(* Action Save NovRAM *)
	IF xAction_SaveNovRAM OR xAction_SaveNovRAMWithoutConfirm THEN
		(* Step saving NovRAM *)
		CASE iStepActionNovRam OF
		(* check NovRAM *)
		1:	xTmp:=	T_NovRAM.T_Ctrle.xDone
					AND NOT(T_NovRAM.T_Ctrle.xExecute)
					AND NOT(T_NovRAM.T_Ctrle.xErr);
			IF xTmp THEN
				(* next Step *)
				iStepActionNovRam :=10;
				xStepActionDone:=FALSE;
			(* activ error *)
			ELSE iStepActionNovRam:=95; END_IF
		(* copy value *)
		10:	IF  xAction_SaveNovRAM THEN
				(* saving with confirmation *)
				TimerAction(IN:=FALSE);
				tTimeOutAction:=T#6s;
				T_Visu.ptrT_ExchgParam^.T_Visu.T_Message.iState:=108;	(* Confirm saving action <Enter>, or escape <Esc> ? *)
				(* next Step *)
				iStepActionNovRam :=20;
			ELSE
				(* next Step *)
				IF xAction_LoadProfileToProcessImage OR xAction_SaveProfileToFile OR xActionDeleteProfile  THEN
					IF xAction_LoadProfileToProcessImage THEN
						T_NovRam.T_Data.T_Standard.T_InfoProcess.iProfile:=T_VisuQVis.ptrT_ExchgParam^.T_StationCommon.T_InfoProcess.iProfile;
						T_NovRam.T_Data.T_Standard.T_InfoProcess.sProfileName:=T_VisuQVis.ptrT_ExchgParam^.T_StationCommon.T_InfoProcess.sProfileName;
					END_IF;
					iStepActionNovRam :=40;
				ELSE
					iStepActionNovRam :=30;
				END_IF;
				(* Display message *)
				T_Visu.ptrT_ExchgParam^.T_Visu.T_Message.iState:=13;	(* Start saving *)
			END_IF;
		(* waiting for saving confirmation key <Enter> or <Esc> *)
		20:	IF RisingEdgeKeyPanel_Enter.Q THEN
			(* Display message *)
				T_Visu.ptrT_ExchgParam^.T_Visu.T_Message.iState:=13;	(* Start saving *)
				(* next step *)
				iStepActionNovRam:=30;
			ELSE
				IF RisingEdgeKeyPanel_Esc.Q THEN iStepActionNovRam:=60; END_IF
				(* An other message has been displayed, stop saving action *)
				IF T_Visu.ptrT_ExchgParam^.T_Visu.T_Message.iState<>108 THEN iStepActionNovRam:=60; END_IF
			END_IF
		30:	T_NovRAM.T_Data.T_ProcessImageData.T_GeometryPara:=T_Visu.ptrT_ExchgParam^.T_GeometryCommon.T_Geometry;
			T_NovRAM.T_Data.T_ProcessImageData.T_PrismPara:=T_Visu.ptrT_ExchgParam^.T_StationCommon.T_PrismPara;
			IF (T_NovRAM.T_Data.T_ProcessImageData.T_PrismPara.bStateInputPrisma = 1) THEN
				T_NovRAM.T_Data.T_ProcessImageData.T_PrismPara.bStateInputPrisma:=0;
			END_IF;
			IF (T_NovRAM.T_Data.T_ProcessImageData.T_PrismPara.bStateInputPrisma = 3) THEN
				T_NovRAM.T_Data.T_ProcessImageData.T_PrismPara.bStateInputPrisma:=2;
			END_IF;
			rCalcMinMaxToolDia:=	rFctCalcMaxToolDiameter(	rDistanceD1:=T_NovRAM.T_Data.T_ProcessImageData.T_PrismPara.rPrismaDistanceD1,
														rDistanceD2:=T_NovRAM.T_Data.T_ProcessImageData.T_PrismPara.rPrismaDistanceD2,
														rAnglePrism:=T_NovRAM.T_Data.T_ProcessImageData.T_PrismPara.rPrismaAngleA);
			T_NovRAM.T_Data.T_ProcessImageData.T_PrismPara.rToolDiameterMax:=rCalcMinMaxToolDia;
			rCalcMinMaxToolDia:=	rFctCalcMinToolDiameter(	rDistanceD1:=T_NovRAM.T_Data.T_ProcessImageData.T_PrismPara.rPrismaDistanceD1,
														rDistanceD2:=T_NovRAM.T_Data.T_ProcessImageData.T_PrismPara.rPrismaDistanceD2,
														rAnglePrism:=T_NovRAM.T_Data.T_ProcessImageData.T_PrismPara.rPrismaAngleA,
														bStateInputPrisma:=T_NovRAM.T_Data.T_ProcessImageData.T_PrismPara.bStateInputPrisma);
			T_NovRAM.T_Data.T_ProcessImageData.T_PrismPara.rToolDiameterMin:=rCalcMinMaxToolDia;
			rCalcPrismaFactor:=	rFctCalcPrismaFactor(	rAnglePrism:=T_NovRAM.T_Data.T_ProcessImageData.T_PrismPara.rPrismaAngleA);
			T_NovRAM.T_Data.T_ProcessImageData.T_PrismPara.rPrismaFactor:=rCalcPrismaFactor;
			T_Visu.ptrT_ExchgParam^.T_StationCommon.T_PrismPara:=T_NovRAM.T_Data.T_ProcessImageData.T_PrismPara;
			T_NovRAM.T_Data.T_Standard.T_TeachINToolLeft:=T_Visu.ptrT_ExchgParam^.T_TeachIn.TParam_ToolLeft;
			T_NovRAM.T_Data.T_Standard.T_TeachINToolCenter:=T_Visu.ptrT_ExchgParam^.T_TeachIn.TParam_ToolCenter;
			T_NovRAM.T_Data.T_Standard.T_TeachINToolRight:=T_Visu.ptrT_ExchgParam^.T_TeachIn.TParam_ToolRight;
			T_NovRAM.T_Data.T_Standard.T_TeachINToolFeeder:=T_Visu.ptrT_ExchgParam^.T_TeachIn.TParam_ToolFeeder;
			T_NovRAM.T_Data.T_Standard.T_TeachINGrindFeeder:=T_Visu.ptrT_ExchgParam^.T_TeachIn.TParam_GrindFeeder;
			T_NovRAM.T_Data.T_Standard.T_AxisPosition:=T_Visu.ptrT_ExchgParam^.T_TeachIn.TParam_AxisPosition;
			T_NovRAM.T_Data.T_Standard.T_MachineConfig.iConfigMachineType:=T_Visu.ptrT_ExchgParam^.T_StationCommon.iConfigMachineType;
			T_NovRAM.T_Data.T_Standard.T_MachineConfig.iConfigAxisType:=T_Visu.ptrT_ExchgParam^.T_StationCommon.iConfigAxisType;
			T_NovRAM.T_Data.T_Standard.T_MachineConfig.iConfigVisuNavigation:=T_Visu.ptrT_ExchgParam^.T_StationCommon.iConfigVisuNavigation;
			T_NovRAM.T_Data.T_Standard.T_MachineConfig.rConfigMaxToolLength:=T_Visu.ptrT_ExchgParam^.T_StationCommon.rConfigMaxToolLength;
			T_NovRAM.T_Data.T_Standard.T_ToolTensionSystem:=T_Visu.ptrT_ExchgParam^.T_StationCommon.T_ParamToolTensionSystem;
			T_NovRAM.T_Data.T_Standard.T_Cyl_ToolTension:=T_Visu.ptrT_ExchgParam^.T_Cylinder.T_ParamToolTension;
			T_NovRAM.T_Data.T_ProcessImageData.T_AutoGeometryPara:=T_Visu.ptrT_ExchgParam^.T_StationCommon.T_AutoGeometryPara;
			T_NovRAM.T_Data.T_ProcessImageData.T_AutoGroovePara:=T_Visu.ptrT_ExchgParam^.T_StationCommon.T_AutoGroovePara;
			T_NovRAM.T_Data.T_ProcessImageData.T_CalibrationPara:=T_Visu.ptrT_ExchgParam^.T_StationCommon.T_CalibrationPara;
			T_NovRAM.T_Data.T_ProcessImageData.T_ProcessPara:=T_Visu.ptrT_ExchgParam^.T_StationCommon.T_ProcessPara;
			(* next Step *)
			iStepActionNovRam :=40;
		(* activ save *)
		40:	T_NovRAM.T_Ctrle.xExecute:=TRUE;
			T_NovRAM.T_Ctrle.iFunction:=2;
			(* next Step *)
			iStepActionNovRam :=50;
			xStepActionDone:=FALSE;
		(* wait save confirmation *)
		50:	IF NOT(xStepActionDone) THEN
				T_NovRAM.T_Ctrle.xExecute:=FALSE;
				(* confirm Step *)
				xStepActionDone:=TRUE;
			ELSE
				IF T_NovRAM.T_Ctrle.xDone THEN
				(* next Step *)
					IF (T_Visu.T_PlcParam.dwActualPage = 430) OR ((T_Visu.T_PlcParam.dwActualPage = 130) AND (T_Visu.T_CtrleAction.iFunction = 1002)) OR
					     ((T_Visu.T_PlcParam.dwActualPage = 470) AND (T_Visu.ptrT_ExchgParam^.T_Config.iEditParam = 410)) THEN
						iStepActionNovRam :=51;
						xOpenMessageBox:=FALSE;
					ELSE
						iStepActionNovRam :=90;
					END_IF;
					xStepActionDone:=FALSE;
				ELSE	IF T_NovRAM.T_Ctrle.xErr THEN
							iStepActionNovRam:=99;
							xStepActionDone:=FALSE;
						END_IF
				END_IF
			END_IF
		(* check first if the Actual position is between the pos and neg SW limit switch *)
		51:	IF (T_Station.THardware.TAxisGrindFeeder.T_LiveValue.lrActualPosition >= T_NovRAM.T_Data.T_ProcessImageData.T_PrismPara.rToolDiameterMin) AND
			     (T_Station.THardware.TAxisGrindFeeder.T_LiveValue.lrActualPosition <= (T_NovRAM.T_Data.T_ProcessImageData.T_PrismPara.rToolDiameterMax + T_NovRAM.T_Data.T_Standard.T_TeachINGrindFeeder.rOffsetSWPosEndSwitch)) THEN
				(* Actual Position is not over the SW limit switches *)
				iStepActionNovRam :=53;
			ELSE
				(* Actual Position is over the SW limit switches *)
				T_Station.THardware.TAxisGrindFeeder.T_CtrleSingle.iFunction:=29;		(* Switch off the SW limit switches, in this case the GrindFeeder will not move automatically *)
				T_Station.THardware.TAxisGrindFeeder.T_CtrleSingle.xExecute:=TRUE;
				iStepActionNovRam :=52;
				xOpenMessageBox:=TRUE;
				tTimeOutAction:=tTimeOutAction + T#9999s;
			END_IF;
		(* Wait end of resettet SW end switch for the GrindFeeder Axis *)
		52:	IF NOT(T_Station.THardware.TAxisGrindFeeder.T_CtrleSingle.xExecute) AND T_Station.THardware.TAxisGrindFeeder.T_CtrleSingle.xDone THEN
				(* set the new position of the GrindFeeder Axis *)
				T_Station.THardware.TAxisGrindFeeder.T_CtrleSingle.rSetPosition:=T_NovRAM.T_Data.T_ProcessImageData.T_PrismPara.rToolDiameterMin;
				T_Station.THardware.TAxisGrindFeeder.T_CtrleSingle.iFunction:=11;
				T_Station.THardware.TAxisGrindFeeder.T_CtrleSingle.xExecute:=TRUE;
				lrActualGrindFeedPosition:=DINT_TO_LREAL(LREAL_TO_DINT(T_Station.THardware.TAxisGrindFeeder.T_LiveValue.lrActualPosition * 100.0)) / 100.0;
				lrToWriteGrindFeedPosition:=DINT_TO_LREAL(LREAL_TO_DINT(T_NovRAM.T_Data.T_ProcessImageData.T_PrismPara.rToolDiameterMin * 100.0)) / 100.0;
				iStepActionNovRam :=53;
			END_IF;
			IF NOT(T_Station.THardware.TAxisGrindFeeder.T_CtrleSingle.xExecute) AND T_Station.THardware.TAxisGrindFeeder.T_CtrleSingle.xErr THEN
				iStepActionNovRam :=98;
			END_IF;
		(* Set SW end switch for the GrindFeeder Axis *)
		53:	IF NOT(T_Station.THardware.TAxisGrindFeeder.T_CtrleSingle.xExecute) AND T_Station.THardware.TAxisGrindFeeder.T_CtrleSingle.xDone THEN
				T_Station.THardware.TAxisGrindFeeder.T_CtrleSingle.iFunction:=28;
				T_Station.THardware.TAxisGrindFeeder.T_CtrleSingle.lrSWNegLimitSwitch:=T_NovRAM.T_Data.T_ProcessImageData.T_PrismPara.rToolDiameterMin;
				T_Station.THardware.TAxisGrindFeeder.T_CtrleSingle.lrSWPosLimitSwitch:=T_NovRAM.T_Data.T_ProcessImageData.T_PrismPara.rToolDiameterMax + T_NovRAM.T_Data.T_Standard.T_TeachINGrindFeeder.rOffsetSWPosEndSwitch;
				T_Station.THardware.TAxisGrindFeeder.T_CtrleSingle.xExecute:=TRUE;
				iStepActionNovRam :=54;
			END_IF;
			IF NOT(T_Station.THardware.TAxisGrindFeeder.T_CtrleSingle.xExecute) AND T_Station.THardware.TAxisGrindFeeder.T_CtrleSingle.xErr THEN
				iStepActionNovRam :=98;
			END_IF;
		(* Wait end of settled SW end switch for the GrindFeeder Axis *)
		54:	IF NOT(T_Station.THardware.TAxisGrindFeeder.T_CtrleSingle.xExecute) AND T_Station.THardware.TAxisGrindFeeder.T_CtrleSingle.xDone THEN
				IF xOpenMessageBox THEN
					xOpenMessageBox:=FALSE;
					iStepActionNovRam :=55;
				ELSE
					iStepActionNovRam :=90;
				END_IF;
			END_IF;
			IF NOT(T_Station.THardware.TAxisGrindFeeder.T_CtrleSingle.xExecute) AND T_Station.THardware.TAxisGrindFeeder.T_CtrleSingle.xErr THEN
				iStepActionNovRam :=98;
			END_IF;
		(* Open MessageBox *)
		55:	T_Visu.ptrT_ExchgParam^.T_FunctionCommon.sMessageBoxLine1:='The prisma value are changed and the actual ';
			T_Visu.ptrT_ExchgParam^.T_FunctionCommon.sMessageBoxLine2:='GrindFeeder position is now over the';
			T_Visu.ptrT_ExchgParam^.T_FunctionCommon.sMessageBoxLine3:='Software limit switches. The actual absolut';
			T_Visu.ptrT_ExchgParam^.T_FunctionCommon.sMessageBoxLine4:='GrindFeeder position: ';
			T_Visu.ptrT_ExchgParam^.T_FunctionCommon.sMessageBoxLine4:=CONCAT(T_Visu.ptrT_ExchgParam^.T_FunctionCommon.sMessageBoxLine4,
																				LREAL_TO_STRING(lrActualGrindFeedPosition));
			T_Visu.ptrT_ExchgParam^.T_FunctionCommon.sMessageBoxLine4:=CONCAT(T_Visu.ptrT_ExchgParam^.T_FunctionCommon.sMessageBoxLine4,'um');
			T_Visu.ptrT_ExchgParam^.T_FunctionCommon.sMessageBoxLine5:='is overwritten with the minimum ';
			T_Visu.ptrT_ExchgParam^.T_FunctionCommon.sMessageBoxLine6:='ToolDiameter: ';
			T_Visu.ptrT_ExchgParam^.T_FunctionCommon.sMessageBoxLine6:=CONCAT(T_Visu.ptrT_ExchgParam^.T_FunctionCommon.sMessageBoxLine6,
																				LREAL_TO_STRING(lrToWriteGrindFeedPosition));
			T_Visu.ptrT_ExchgParam^.T_FunctionCommon.sMessageBoxLine6:=CONCAT(T_Visu.ptrT_ExchgParam^.T_FunctionCommon.sMessageBoxLine6,'um');
			T_Visu.ptrT_ExchgParam^.T_FunctionCommon.xOpenOverlayMessageBox:=TRUE;
			iStepActionNovRam :=56;
		(* Wait cofirming of the messagebox *)
		56:	IF NOT(T_Visu.ptrT_ExchgParam^.T_FunctionCommon.xOpenOverlayMessageBox) THEN
				iStepActionNovRam :=90;
			END_IF;
			IF T_Visu.T_CtrleAction.xDone THEN
				T_Visu.ptrT_ExchgParam^.T_FunctionCommon.xOpenOverlayMessageBox:=FALSE;
				xAction_SaveNovRAM:=FALSE;
				xAction_SaveNovRAMWithoutConfirm:=FALSE;
				T_Visu.ptrT_ExchgParam^.T_Visu.T_Message.iState:=0;
			END_IF;
		(* Reset settled value *)
		60:	xResetParaListValue:=TRUE;
			iStepActionNovRam:=70;
		70:	IF NOT(xResetParaListValue) THEN
				iStepActionNovRam:=90;
			END_IF;
		(* no code, waiting timeout *)
		89:	IF TimerAction.Q THEN iStepActionNovRam:=90; END_IF
		(* save done *)
		90:	T_Visu.ptrT_ExchgParam^.T_Visu.T_Message.iState:=0;
			T_Visu.T_CtrleAction.xDone:=TRUE;
			T_Visu.T_CtrleAction.xNotReady:=FALSE;
			T_Visu.T_CtrleAction.xErr:=FALSE;
			T_Visu.T_CtrleAction.udiErrorID:=0;
			xAction_SaveNovRAM:=FALSE;
			xAction_SaveNovRAMWithoutConfirm:=FALSE;
			T_Visu.ptrT_ExchgParam^.T_FunctionCommon.xOpenOverlayMessageBox:=FALSE;
		(* NovRAM not ready *)
		95:	TimerNotReady(IN:=TRUE);
			xAction_SaveNovRAM:=FALSE;
			xAction_SaveNovRAMWithoutConfirm:=FALSE;
			T_Visu.ptrT_ExchgParam^.T_FunctionCommon.xOpenOverlayMessageBox:=FALSE;
		(* error *)
		98:	T_Visu.ptrT_ExchgParam^.T_StationCommon.wState:=T_Visu.ptrT_ExchgParam^.T_StationCommon.wState AND 16#BF;
			T_Visu.T_CtrleAction.xDone:=TRUE;
			T_Visu.T_CtrleAction.xNotReady:=FALSE;
			IF (T_Station.THardware.TAxisGrindFeeder.T_Config_Gen.iTyp <> 0) THEN
				diErrorNr:=(T_Station.THardware.TAxisGrindFeeder.T_Config_Gen.iTyp * 1000000) + T_Station.THardware.TAxisGrindFeeder.T_CtrleSingle.udiErrorID;
			ELSE
				diErrorNr:=0;
			END_IF;
			FBErrorMessage(	diErrorNr:=diErrorNr,
							T_ErrorList:=T_ErrorList);
			T_Visu.ptrT_ExchgParam^.T_Visu.T_Message.sDynamicTextEnglish:=FBErrorMessage.sErrorTextEnglish;
			T_Visu.ptrT_ExchgParam^.T_Visu.T_Message.sDynamicTextDeutsch:=FBErrorMessage.sErrorTextDeutsch;
			T_Visu.ptrT_ExchgParam^.T_Visu.T_Message.sDynamicTextFrancais:=FBErrorMessage.sErrorTextFrancais;
			T_Visu.ptrT_ExchgParam^.T_SafetyCtrl.xSetForceError:=TRUE;
			T_Visu.ptrT_ExchgParam^.T_SafetyCtrl.diSetForceErrorNr:=diErrorNr;
			T_Visu.T_CtrleAction.xErr:=FALSE;
			T_Visu.T_CtrleAction.udiErrorID:=0;
			T_Station.THardware.TAxisGrindFeeder.T_CtrleSingle.iFunction:=1;
			T_Station.THardware.TAxisGrindFeeder.T_CtrleSingle.xExecute:=TRUE;
			xAction_SaveNovRAM:=FALSE;
			xAction_SaveNovRAMWithoutConfirm:=FALSE;
			T_Visu.ptrT_ExchgParam^.T_FunctionCommon.xOpenOverlayMessageBox:=FALSE;
		(* error *)
		99:	T_Visu.T_CtrleAction.xDone:=FALSE;
			T_Visu.T_CtrleAction.xNotReady:=FALSE;
			T_Visu.T_CtrleAction.xErr:=TRUE;
			T_Visu.T_CtrleAction.udiErrorID:=16#F0000 + T_Visu.T_CtrleAction.iFunction;
			xAction_SaveNovRAM:=FALSE;
			xAction_SaveNovRAMWithoutConfirm:=FALSE;
			T_Visu.ptrT_ExchgParam^.T_FunctionCommon.xOpenOverlayMessageBox:=FALSE;
		END_CASE
	END_IF;

(* Delete Profile *)
	IF xActionDeleteProfile THEN
		(* Step delete profile *)
		CASE iStepAction OF
		(* Profile number could not be 1 *)
		1:	IF T_Visu.ptrT_ExchgParam^.T_ProfileCommon.T_Id.iNumber < 2 THEN
				 tTimeOutAction:=TimerAction.ET+T#2s;
				T_Visu.ptrT_ExchgParam^.T_Visu.T_Message.iState:=27;	(* Default profile can't be deleted *)
				iStepAction:=10;
			ELSIF T_Visu.ptrT_ExchgParam^.T_StationCommon.T_InfoProcess.iProfile = T_Visu.ptrT_ExchgParam^.T_ProfileCommon.T_Id.iNumber THEN
				tTimeOutAction:=TimerAction.ET+T#2s;
				T_Visu.ptrT_ExchgParam^.T_Visu.T_Message.iState:=28;	(* Load profile can't be deleted *)
				iStepAction:=10;
			ELSE iStepAction:=20; END_IF
		(* no code, waiting timeout *)
		10:	IF TimerAction.Q THEN xActionDeleteProfile:=FALSE; END_IF;
		(* Display message to ask for confirmation *)
		20:	T_Visu.ptrT_ExchgParam^.T_Visu.T_Message.iState:=117;	(* Confirm delete profile <Enter>, or escape <Esc> ? *)
			(* next step *)
			iStepAction:=30;
		(* waiting for key <Enter> or <Esc> *)
		30:	IF RisingEdgeKeyPanel_Enter.Q THEN
				(* Display message deleting *)
				T_Visu.ptrT_ExchgParam^.T_Visu.T_Message.iState:=29;	(* Start deleting *)
				(* next step *)
				iStepAction:=40;
			ELSE
				IF RisingEdgeKeyPanel_Esc.Q THEN iStepAction:=90; END_IF
				(* An other message has been displayed, stop import/export action *)
				IF T_Visu.ptrT_ExchgParam^.T_Visu.T_Message.iState<>117 THEN iStepAction:=90; END_IF
			END_IF;
		(* Init. deleting profile file *)
		40:	IF T_NovRam.T_Data.T_IDProfileStation[T_Visu.ptrT_ExchgParam^.T_ProfileCommon.T_Id.iNumber].sName <> '' THEN
				sTmp:='\Hard Disk\Machine450\Profile\';
				sTmp:=CONCAT(sTmp,T_NovRam.T_Data.T_IDProfileStation[T_Visu.ptrT_ExchgParam^.T_ProfileCommon.T_Id.iNumber].sName);
				T_HDD.T_File.sPathAndFileName:=CONCAT(sTmp,'.txt');
				(* activ delete file *)
				T_HDD.T_Ctrle.xExecute:=TRUE;
				T_HDD.T_Ctrle.iFunction:=5;
				iStepAction:=50;
			(* Display info message 'file does not exists *)
			ELSE
				T_Visu.ptrT_ExchgParam^.T_Visu.T_Message.iState:=11;
				(* next step *)
				iStepAction:=55;
				xStepActionDone:=FALSE;
				tTimeOutAction:=TimerAction.ET+T#2s;
			END_IF
		50:	IF NOT T_HDD.T_Ctrle.xExecute AND (T_HDD.T_Ctrle.xDone OR T_HDD.T_Ctrle.xErr) THEN
				T_HDD.T_Ctrle.xReset:=T_HDD.T_Ctrle.xErr;
				(* Profile will be erased from the profile list *)
				T_NovRam.T_Data.T_IDProfileStation[T_Visu.ptrT_ExchgParam^.T_ProfileCommon.T_Id.iNumber].sName:='';
				xUpdateProfileList:=TRUE;
				IF T_HDD.T_Ctrle.xErr THEN
					(* Display info message 'file does not exists *)
					T_Visu.ptrT_ExchgParam^.T_Visu.T_Message.iState:=11;
					(* next step *)
					iStepAction:=52;
					xStepActionDone:=FALSE;
					(* use tmp timer to diplay message *)
					TimerONTmp(IN:=FALSE);
					TimerONTmp.PT:=T#2s;
				ELSE
					(* next step *)
					iStepAction:=70;
					xStepActionDone:=FALSE;
				END_IF;
			END_IF
		(* Wait delay timer *)
		52:	IF TimerONTmp.Q THEN
				T_Visu.ptrT_ExchgParam^.T_Visu.T_Message.iState:=0;
				(* next step *)
				iStepAction:=70;
			END_IF
		(* delay time out *)
		55:	IF TimerAction.Q THEN xActionDeleteProfile:=FALSE; END_IF
		(* active saving data NovRAM *)
		70:	T_Visu.ptrT_ExchgParam^.T_ProfileCommon.T_Id.sName:='';
			xAction_SaveNovRAMWithoutConfirm:=TRUE;
			iStepActionNovRam:=1;
			(* next step *)
			iStepAction:=80;
		(* waiting confirm saving NovRAM action *)
		80:	IF NOT xAction_SaveNovRAMWithoutConfirm THEN iStepAction:=90; END_IF
		(* save done *)
		90:	T_Visu.ptrT_ExchgParam^.T_Visu.T_Message.iState:=0;
			T_Visu.T_CtrleAction.xDone:=TRUE;
			T_Visu.T_CtrleAction.xNotReady:=FALSE;
			T_Visu.T_CtrleAction.xErr:=FALSE;
			T_Visu.T_CtrleAction.udiErrorID:=0;
			xActionDeleteProfile:=FALSE;
		(* Action not ready *)
		95:	TimerNotReady(IN:=TRUE);
			xActionDeleteProfile:=FALSE;
		(* error *)
		99:	T_Visu.T_CtrleAction.xDone:=FALSE;
			T_Visu.T_CtrleAction.xNotReady:=FALSE;
			T_Visu.T_CtrleAction.xErr:=TRUE;
			T_Visu.T_CtrleAction.udiErrorID:=16#F1000 + T_Profile.T_Ctrle.iFunction;
			xActionDeleteProfile:=FALSE;
		END_CASE;
	END_IF;

(* Action start process machine or station *)
	IF xActionProcMachine OR xActionProcStation THEN
		(* Step process machine *)
		CASE iStepAction OF
		(* check process state *)
		1:	xTmp:=	T_Process.xEnable AND
					T_Process.xEnd AND
					T_Process.xRdy AND
					NOT(T_Process.xStop) AND
					NOT(T_Process.xStopCycle) AND
					NOT(T_Process.xError);
			(* next step *)
			IF NOT(xTmp) THEN
				iStepAction:=95;
			ELSE IF xActionProcMachine THEN iStepAction:=10; ELSE iStepAction:=20; END_IF
			END_IF
		(* check process number and start process machine *)
		10:	CASE T_Process.iFunctNr OF
			(* process available *)
			(*	10=Process AutoGeometry
				20=Process AutoGroove
				30=Process Reference
			*)
			10,20,30:	T_Visu.T_CtrleProcess.iFunction:=1;
						T_Visu.T_CtrleProcess.xExecute:=TRUE;
						iStepAction:=90;
			(* unknown process *)
			ELSE	iStepAction:=95;
			END_CASE
			(* next step *)
			xStepActionDone:=FALSE;
		(* check process number and start process station *)
		20:	CASE T_Process.iFunctNr OF
			(* process available *)
			(*	40=ToolCalibration
			*)
			40:	T_Visu.T_CtrleProcess.iFunction:=2;
				T_Visu.T_CtrleProcess.xExecute:=TRUE;
				iStepAction:=90;
			(* unknown process *)
			ELSE
				iStepAction:=95;
			END_CASE
			(* next step *)
			xStepActionDone:=FALSE;
		(* Display message, waiting timeout *)
		89:	IF TimerAction.Q THEN
				(* init. trigger FB_CtrleButton Start/Stop *)
				T_Visu.ptrT_ExchgParam^.T_Machine.T_Process.wState:=16#0;
				(* action done *)
				iStepAction:=90;
			END_IF
		(* action done *)
		90:	T_Visu.T_CtrleAction.xDone:=TRUE;
			T_Visu.T_CtrleAction.xNotReady:=FALSE;
			T_Visu.T_CtrleAction.xErr:=FALSE;
			T_Visu.T_CtrleAction.udiErrorID:=0;
			xActionProcMachine:=FALSE;
			xActionProcStation:=FALSE;
		(* cylinder not ready *)
		95:	TimerNotReady(IN:=TRUE);
			xActionProcMachine:=FALSE;
			xActionProcStation:=FALSE;
		(* error *)
		99:	T_Visu.T_CtrleAction.xDone:=FALSE;
			T_Visu.T_CtrleAction.xNotReady:=FALSE;
			T_Visu.T_CtrleAction.xErr:=TRUE;
			T_Visu.T_CtrleAction.udiErrorID:=16#F0000 + T_Visu.T_CtrleAction.iFunction;
			xActionProcMachine:=FALSE;
			xActionProcStation:=FALSE;
		END_CASE
	END_IF

(* Manage process execution *)
	(* ...done *)
	RisingEdgeProcessDone(CLK:=T_Visu.T_CtrleProcess.xDone);
	IF RisingEdgeProcessDone.Q THEN
		IF NOT(T_StartUp.T_State.xBlockChangeMovementVisu) THEN
			IF T_Visu.T_CtrleProcess.iFunction <> 0 AND T_Visu.ptrT_ExchgParam^.T_Visu.T_Message.iState = 0 THEN
			(* call confirmation message *)
				IF NOT xStopImmediatly THEN
					IF (T_Visu.T_PlcParam.dwActualPage = 110) THEN
						T_Visu.ptrT_ExchgParam^.T_Visu.T_Message.iState:=22;
					END_IF;
					(*T_Visu.ptrT_ExchgParam^.T_Visu.T_Message.iState
						:=iFctReturnConfMessage(iNumAction:=T_Process.iFunctNr+1100);*);
				(* Display message 'Process is aborded' *)
				ELSE T_Visu.ptrT_ExchgParam^.T_Visu.T_Message.iState:=9; END_IF
			END_IF
		END_IF;
	END_IF
	(* ...error *)
	RisingEdgeProcessError(CLK:=T_Visu.T_CtrleProcess.xErr);
	IF RisingEdgeProcessError.Q THEN
	(* call function bloc action error *)
		IF NOT(T_StartUp.T_State.xBlockChangeMovementVisu) THEN
			(*
			fbQvisError(	udiActionError:=T_Visu.T_CtrleProcess.udiErrorID,
						T_Message:=T_Visu.ptrT_ExchgParam^.T_Visu.T_Message);
			*);
		END_IF;
		(* Init. variable *)
		T_Visu.T_CtrleProcess.xExecute:=FALSE;
		T_Visu.T_CtrleProcess.xDone:=TRUE;
		T_Visu.T_CtrleProcess.xErr:=FALSE;
		T_Visu.T_CtrleProcess.udiErrorID:=0;
		(*iStepProcess:=1;*)
		(*xStepProcessDone:=FALSE;*)
	END_IF
	(* ...reset *)
	RisingEdgeResetProcess(CLK:=T_Visu.T_CtrleProcess.xReset);
	IF RisingEdgeResetProcess.Q THEN
		(* Init. variable *)
		T_Visu.T_CtrleProcess.xExecute:=FALSE;
		T_Visu.T_CtrleProcess.xDone:=TRUE;
		T_Visu.T_CtrleProcess.xErr:=FALSE;
		T_Visu.T_CtrleProcess.udiErrorID:=0;
		(*iStepProcess:=1;*)
		(*xStepProcessDone:=FALSE;*)
		(* Release process *)
		T_Visu.T_CtrleProcess.xReset:=FALSE;
	END_IF
	RisingEdgeExecuteProcess(CLK:=T_Visu.T_CtrleProcess.xExecute);
	IF RisingEdgeExecuteProcess.Q THEN
		(* Release execution *)
		T_Visu.T_CtrleProcess.xExecute:=FALSE;
		CASE T_Visu.T_CtrleProcess.iFunction OF
		(* Process machine *)
		1:	xProcessMachine:=TRUE;
		(* Process station *)
		2:	xProcessStation:=TRUE;
		(* process not implemented *)
		ELSE	T_Visu.T_CtrleProcess.xDone:=FALSE;
				T_Visu.T_CtrleProcess.xErr:=TRUE;
				T_Visu.T_CtrleProcess.udiErrorID:=16#E000;
				(* exit FB *)
				RETURN;
		END_CASE
		(* Init. variable *)
		T_Visu.T_CtrleProcess.xDone:=FALSE;
		T_Visu.T_CtrleProcess.xErr:=FALSE;
		T_Visu.T_CtrleProcess.udiErrorID:=0;
		iStepProcess:=1;
		xStepProcessDone:=FALSE;
		(* exit FB *)
		RETURN;
	END_IF

(* Process machine *)
	IF xProcessMachine OR xProcessStation THEN
		CASE iStepProcess OF
		(* check process number and start process machine *)
		1:	T_Process.xStart:=TRUE;
			iStepProcess:=10;
			IF (T_Visu.T_PlcParam.dwActualPage = 10) THEN
				T_Visu.ptrT_ExchgParam^.T_SafetyCtrl.bStateAutoGeometry:=2;
			ELSIF (T_Visu.T_PlcParam.dwActualPage = 20) THEN
				T_Visu.ptrT_ExchgParam^.T_SafetyCtrl.bStateAutoGroove:=2;
			ELSIF (T_Visu.T_PlcParam.dwActualPage = 30) THEN
				T_Visu.ptrT_ExchgParam^.T_SafetyCtrl.bStateReference:=2;
			ELSIF (T_Visu.T_PlcParam.dwActualPage = 110) THEN
				T_Visu.ptrT_ExchgParam^.T_SafetyCtrl.bStateToolCalibration:=2;
			END_IF;
			(* next step *)
			xStepProcessDone:=FALSE;
		(* wait confirmation *)
		10:	IF NOT(xStepProcessDone) THEN
			(* release execution *)
				T_Process.xStart:=FALSE;
				xStepProcessDone:=TRUE;
				IF T_Visu.ptrT_ExchgParam^.T_StationCommon.T_AutoGeometryPara.xWarmUp THEN
					xWarmUpMessageActiv:=TRUE;
					xWarmUpMessageDone:=TRUE;
				END_IF;
			ELSE
				IF T_Process.xEnd THEN
					(* action done *)
					iStepProcess:=90;
					xStepProcessDone:=FALSE;
				ELSE
					IF T_Visu.ptrT_ExchgParam^.T_StationCommon.T_AutoGeometryPara.xWarmUp AND xWarmUpMessageActiv THEN
						T_Visu.ptrT_ExchgParam^.T_Visu.T_Message.iState:=124;	(* WarmUp cycle activ *)
						xWarmUpMessageActiv:=FALSE;
					END_IF;
					IF (T_Visu.ptrT_ExchgParam^.T_Visu.T_Message.iState=124                                                 )	AND
					     NOT(T_Visu.ptrT_ExchgParam^.T_StationCommon.T_AutoGeometryPara.xWarmUp) 	AND
					     xWarmUpMessageDone 															THEN
						T_Visu.ptrT_ExchgParam^.T_Visu.T_Message.iState:=125;	(*WarmUp cycle time arrived. <Press StopButton>*)
						xWarmUpMessageDone:=FALSE;
					END_IF;
					IF T_Process.xError THEN
						(* action error *)
						iStepProcess:=99;
						xStepProcessDone:=FALSE;
						IF xProcessMachine THEN
							T_Visu.ptrT_ExchgParam^.T_TouchScreenBtPanel.iStateBtLeft:=0;
							IF(T_Process.iFunctNr = 10) THEN
								IF (T_Visu.T_PlcParam.dwActualPage <> 10) THEN
									T_Visu.T_PlcParam.dwSetNewPage:=10;
									T_Visu.T_CtrleVisu.iFunction:=1;
									T_Visu.T_CtrleVisu.xExecute:=TRUE;
								END_IF;
							END_IF;
							IF(T_Process.iFunctNr = 20) THEN
								IF (T_Visu.T_PlcParam.dwActualPage <> 20) THEN
									T_Visu.T_PlcParam.dwSetNewPage:=20;
									T_Visu.T_CtrleVisu.iFunction:=1;
									T_Visu.T_CtrleVisu.xExecute:=TRUE;
								END_IF;
							END_IF;
							IF(T_Process.iFunctNr = 30) THEN
								IF (T_Visu.T_PlcParam.dwActualPage <> 30) THEN
									T_Visu.T_PlcParam.dwSetNewPage:=30;
									T_Visu.T_CtrleVisu.iFunction:=1;
									T_Visu.T_CtrleVisu.xExecute:=TRUE;
								END_IF;
							END_IF;
							IF(T_Process.iFunctNr = 40) THEN
								IF (T_Visu.T_PlcParam.dwActualPage <> 110) THEN
									T_Visu.T_PlcParam.dwSetNewPage:=110;
									T_Visu.T_CtrleVisu.iFunction:=1;
									T_Visu.T_CtrleVisu.xExecute:=TRUE;
								END_IF;
							END_IF;
						END_IF;
					END_IF
				END_IF
				IF NOT(T_TwinSafeOut.QxContactor_K3) OR NOT(T_TwinSafeOut.QxContactor_K4) THEN
					(*T_Process.xEnable:=FALSE;*)
					(*iStepProcess:=21;*)
					iStepProcess:=99;
					RETURN;
				END_IF;
			END_IF
		21:	IF NOT(T_Process.xEnd) THEN
				T_Process.xEnable:=TRUE;
				iStepProcess:=22;
			ELSE
				T_Process.xEnable:=FALSE;
			END_IF;
		22:	IF T_Process.xEnd THEN
				T_Visu.T_CtrleProcess.xDone:=TRUE;
				T_Visu.T_CtrleProcess.xErr:=FALSE;
				T_Visu.T_CtrleProcess.udiErrorID:=0;
				xProcessMachine:=FALSE;
				xProcessStation:=FALSE;
			END_IF;
		(* call page *)
		30:	T_Visu.T_PlcParam.dwSetNewPage:=dwPageNrProcessStart;
			T_Visu.T_CtrleVisu.iFunction:=2;
			T_Visu.T_CtrleVisu.xExecute:=TRUE;
			(* next step *)
			iStepProcess:=90;
		(* process done *)
		90:	IF NOT(T_Visu.T_CtrleVisu.xExecute) AND T_Visu.T_CtrleVisu.xDone THEN
				T_StartUp.T_State.xBlockChangeMovementVisu:=FALSE;
				IF (T_Visu.T_PlcParam.dwActualPage = 10) THEN
					T_Visu.ptrT_ExchgParam^.T_SafetyCtrl.bStateAutoGeometry:=1;
				ELSIF (T_Visu.T_PlcParam.dwActualPage = 20) THEN
					T_Visu.ptrT_ExchgParam^.T_SafetyCtrl.bStateAutoGroove:=1;
				ELSIF (T_Visu.T_PlcParam.dwActualPage = 30) THEN
					T_Visu.ptrT_ExchgParam^.T_SafetyCtrl.bStateReference:=1;
				ELSIF (T_Visu.T_PlcParam.dwActualPage = 110) THEN
					T_Visu.ptrT_ExchgParam^.T_SafetyCtrl.bStateToolCalibration:=1;
				END_IF;
				IF xProcessMachine THEN
					IF NOT(T_StartUp.T_State.xBlockChangeMovementVisu) THEN
						T_StartUp.T_Ctrle.xExecute:=TRUE;
						T_StartUp.T_Ctrle.iFunction:=11;	(* Acitvate Info Message Overlay *)
						IF (T_Process.iFunctNr = 30) THEN
							(* THE REFERENCE DRIVE  IS COMPLEATED! *)
							(* CONFIRM THIS MESSAGE AND *)
							(* THE MACHINE WILL BE READY! *)
							(*  *)
							T_StartUp.T_Ctrle.iMsgNumber:=3;
						END_IF;
						IF (T_Process.iFunctNr = 10) OR (T_Process.iFunctNr = 20) THEN
							(* THE  AUTO MODE CYCLE IS COMPLEATED! *)
							(* CONFIRM THIS MESSAGE AND *)
							(* THE MACHINE WILL BE READY! *)
							(*  *)
							T_StartUp.T_Ctrle.iMsgNumber:=2;
						END_IF;
					END_IF;
				END_IF;
				T_Visu.T_CtrleProcess.xDone:=TRUE;
				T_Visu.T_CtrleProcess.xErr:=FALSE;
				T_Visu.T_CtrleProcess.udiErrorID:=0;
				xProcessMachine:=FALSE;
				xProcessStation:=FALSE;
			END_IF;
		(* error *)
		99:	IF NOT(T_Visu.T_CtrleVisu.xExecute) AND T_Visu.T_CtrleVisu.xDone THEN
				T_StartUp.T_State.xBlockChangeMovementVisu:=FALSE;
				IF xProcessMachine THEN
					T_StartUp.T_Ctrle.xExecute:=TRUE;
					T_StartUp.T_Ctrle.iFunction:=10;	(* Activate Error Message Overlay *)
					IF (T_Process.iFunctNr = 30) THEN
						(* DURING MACHINE REFERENCE PROC. *)
						(* AN ERROR HAS OCCURRED *)
						(* PLEASE CONFIRM  AND CHECK *)
						(* THE ACCORDING ERROR *)
						T_StartUp.T_Ctrle.iMsgNumber:=14;
					END_IF;
					IF (T_Process.iFunctNr = 10) OR (T_Process.iFunctNr = 20) THEN
						(* DURING THE AUTO MODE *)
						(* AN ERROR HAS OCCURRED *)
						(* PLEASE CONFIRM AND CHECK *)
						(* THE ACCORDING ERROR *)
						T_StartUp.T_Ctrle.iMsgNumber:=13;
					END_IF;
				END_IF;
				T_Visu.T_CtrleProcess.xDone:=FALSE;
				T_Visu.T_CtrleProcess.xErr:=TRUE;
				T_Visu.T_CtrleProcess.udiErrorID:=16#E0000 + T_Visu.T_CtrleProcess.iFunction;
				xProcessMachine:=FALSE;
				xProcessStation:=FALSE;
			END_IF;
		END_CASE
	END_IF

(* Stop process *)
	IF xStopProcess OR xAction_StopCycle THEN
		(* Set stop process *)
		CASE iStepAction OF
		(* check process state and stop process if possible *)
		1:	IF NOT xStopButton THEN
				xTmp:=	T_Process.xRdy
						AND NOT T_Process.xStop
						AND NOT T_Process.xStopCycle
						AND NOT T_Process.xEnd
						AND NOT T_Process.xError
						AND NOT T_Process.xAbord;
				IF xStopProcess AND T_Process.xStopCycle AND NOT(T_Process.xEnd) AND NOT(T_Process.xError) AND NOT(T_Process.xStop) THEN
					xTmp:=TRUE;
				END_IF;
				IF xAction_StopCycle THEN
					IF (T_NovRAM.T_Data.T_ProcessImageData.T_AutoGeometryPara.iCycleGeometry <= 1) THEN
						xTmp:=FALSE;
					END_IF;
				END_IF;
				IF xTmp THEN
					IF xStopProcess THEN
					(* activ stop immediat *)
						T_Process.xStop:=TRUE;
						T_Process.xStopCycle:=NOT T_Process.xStop;
						xBlockConfirmMessage:=TRUE;
						(* Display info message *)
						T_Visu.ptrT_ExchgParam^.T_Visu.T_Message.iState:=122;	(* Stop process immediately *)
						(* set variable *)
						xStopImmediatly:=TRUE;
						(* next step *)
						iStepAction:=20;
					END_IF;
					IF xAction_StopCycle THEN
						T_Process.xStopCycle:=TRUE;
						T_Process.xStop:=NOT T_Process.xStopCycle;
						xBlockConfirmMessage:=TRUE;
						(* Display message *)
						T_Visu.ptrT_ExchgParam^.T_Visu.T_Message.iState:=103;	(* Process will be stopped at the end of the cycle *)
						(* next step *)
						iStepAction:=20;
					END_IF;
				(* not ready to execute stop *)
				ELSE iStepAction:=95; END_IF
			END_IF
			IF T_Process.xError THEN iStepAction:=99; END_IF
		(* waiting function done *)
		20:	IF T_Visu.T_CtrleVisu.xDone THEN
				IF (T_Visu.T_PlcParam.dwActualPage = 10) OR (T_Visu.T_PlcParam.dwActualPage = 20) OR (T_Visu.T_PlcParam.dwActualPage = 30) OR (T_Visu.T_PlcParam.dwActualPage = 110) THEN
					xWaitStopEnd:=xStopProcess;
					xWaitStopCycleEnd:=xAction_StopCycle;
					iStepWaitStopEnd:=1;
				ELSE
					xWaitStopEnd:=FALSE;
					xWaitStopCycleEnd:=FALSE;
				END_IF;
				(* no activ station for machine level *)
				IF T_Visu.T_PlcParam.dwActualPage < 100 THEN
					T_Visu.ptrT_ExchgParam^.T_TouchScreenBtPanel.iStateBtLeft:=0;
				END_IF
				(* next step *)
				iStepAction:=90;
			END_IF
			IF T_Visu.T_CtrleVisu.xErr THEN iStepAction:=99; END_IF
		(* End function *)
		90:	T_Visu.T_CtrleAction.xDone:=TRUE;
			T_Visu.T_CtrleAction.xErr:=FALSE;
			T_Visu.T_CtrleAction.udiErrorID:=16#0;
			xStopProcess:=FALSE;
			xAction_StopCycle:=FALSE;
		(* not ready *)
		95:	TimerNotReady(IN:=TRUE);
			xStopProcess:=FALSE;
			xAction_StopCycle:=FALSE;
		(* Error *)
		99:	T_Visu.T_CtrleAction.xDone:=FALSE;
			T_Visu.T_CtrleAction.xErr:=TRUE;
			T_Visu.T_CtrleAction.udiErrorID:=16#F0000 + T_Visu.T_CtrleAction.iFunction;
			xStopProcess:=FALSE;
			xAction_StopCycle:=FALSE;
		END_CASE
	END_IF

(* Wait End of Stop Machine Process *)
	IF xWaitStopEnd OR xWaitStopCycleEnd THEN
		CASE iStepWaitStopEnd OF
			1:	IF T_Process.xEnd THEN
					iStepWaitStopEnd:=10;
				END_IF;
				IF T_Process.xError THEN
					xWaitStopEnd:=FALSE;
					xWaitStopCycleEnd:=FALSE;
					iStepWaitStopEnd:=1;
				END_IF;
			10:	IF NOT(T_Visu.T_CtrleVisu.xExecute) AND T_Visu.T_CtrleVisu.xDone THEN
					T_Visu.ptrT_ExchgParam^.T_Visu.T_Message.iState:=0;
					IF (T_Process.iFunctNr = 30) THEN
						T_StartUp.T_Ctrle.xExecute:=TRUE;
						T_StartUp.T_Ctrle.iFunction:=11;	(* Acitvate Info Message Overlay *)
						(* THE REFERENCE DRIVE IS STOPPED! *)
						(* CONFIRM THIS MESSAGE AND *)
						(* THE MACHINE WILL BE READY! *)
						(*  *)
						T_StartUp.T_Ctrle.iMsgNumber:=5;
					END_IF;
					IF (T_Process.iFunctNr = 10) OR (T_Process.iFunctNr = 20) THEN
						T_StartUp.T_Ctrle.xExecute:=TRUE;
						T_StartUp.T_Ctrle.iFunction:=11;	(* Acitvate Info Message Overlay *)
						(* THE AUTO MODE CYCLE IS STOPPED! *)
						(* CONFIRM THIS MESSAGE AND *)
						(* THE MACHINE WILL BE READY! *)
						(*  *)
						T_StartUp.T_Ctrle.iMsgNumber:=4;
					END_IF;
					xWaitStopEnd:=FALSE;
					xWaitStopCycleEnd:=FALSE;
					iStepWaitStopEnd:=1;
				END_IF;
		END_CASE;
	END_IF;
(************************************************************************************************************************************************************************)
(***************                                             end for the section for defined function of the visualisation interface                                                ********************)
(************************************************************************************************************************************************************************)

(************************************************************************************************************************************************************************)
(***************                                                 management for the changement of a page on the visualisation                                                 ********************)
(************************************************************************************************************************************************************************)
(* waiting for changing page *)
	RisingEdgeExecute(CLK:=T_Visu.T_CtrleVisu.xExecute);
	IF RisingEdgeExecute.Q THEN
		CASE T_Visu.T_CtrleVisu.iFunction OF
		(* change page *)
		1:	xChangePage:=TRUE;
			dwInCount_QVisCmd:=T_CtrleQVis.dwInCount;
		ELSE
		(* function not implemented *)
			T_Visu.T_CtrleVisu.xDone:=FALSE;
			T_Visu.T_CtrleVisu.xErr:=TRUE;
			T_Visu.T_CtrleVisu.udiErrorID:=16#F000;
		END_CASE
		(* Init. variable *)
		T_Visu.T_CtrleVisu.xDone:=FALSE;
		T_Visu.T_CtrleVisu.xErr:=FALSE;
		T_Visu.T_CtrleVisu.udiErrorID:=0;
		(* exit FB *)
		RETURN;
	END_IF

(* waiting for changing page from the PLC *)
	IF xChangePage THEN
		IF dwInCount_QVisCmd = T_CtrleQVis.dwInCount THEN
			(* Init. command *)
			T_CtrleQVis.dwInCommand:=1;
			T_CtrleQVis.dwInQVisCtrlAddress:=ADR(T_CtrleQVis);
			T_CtrleQVis.dwInParameterAddress:=ADR(T_Visu.T_PlcParam.dwSetNewPage);
			(* start command *)
			T_CtrleQVis.dwInCount:=T_CtrleQVis.dwInCount+1;
		ELSE
			IF T_CtrleQVis.dwInCount = T_CtrleQVis.dwOutCount THEN
			(* command done *)
				T_Visu.T_CtrleVisu.xExecute:=FALSE;
				IF T_CtrleQVis.diOutStatus = 0 THEN
				(* command done without error *)
					T_Visu.T_CtrleVisu.xDone:=TRUE;
					T_Visu.T_CtrleVisu.xErr:=FALSE;
					T_Visu.T_CtrleVisu.udiErrorID:=0;
					(* update value *)
					T_Visu.T_PlcParam.dwPreviousPage:=T_Visu.T_PlcParam.dwActualPage;
					T_Visu.T_PlcParam.dwActualPage:=T_Visu.T_PlcParam.dwSetNewPage;
					IF (T_Visu.T_PlcParam.dwActualPage = 10) THEN
						wNormalLayerActivTask:=1;
						wNormalLayerActivPage:=10;
					END_IF;
				ELSE
				(* command done with error *)
					T_Visu.T_CtrleVisu.xDone:=FALSE;
					T_Visu.T_CtrleVisu.xErr:=TRUE;
					T_Visu.T_CtrleVisu.udiErrorID:=16#F400 + DINT_TO_UDINT(T_CtrleQVis.diOutStatus);
				END_IF
				(* reset variable 'xChangePage' *)
				xChangePage:=FALSE;
			END_IF
		END_IF
	END_IF
END_FUNCTION_BLOCK

(* POU PRG_VISU_LAYER5/FB_VISU/FBQVIS_INITPAGE, ST *)
FUNCTION_BLOCK FBQVIS_INITPAGE
VAR_INPUT
END_VAR
VAR_OUTPUT
END_VAR
VAR_IN_OUT
	T_Visu:ST_QVIS;			(* data structure of the visualisation *)
END_VAR
VAR
(* pointer *)
	ptrConfigPage: POINTER TO ST_CONFIGPAGE;
(* variable *)
	iIndexPage:INT;
	iPageNumber:INT;
(* variable Tmp *)
	i:INT;
END_VAR
(****************************************************************************************************************************************************)
(***********                    This Functionblock init all the defined page in QVis for the hole page management                            ************)
(****************************************************************************************************************************************************)
(* init. index array *)
FOR i:=0 TO 999 DO
	T_Visu.T_PageIndex[i].iIndexConfigPage:=0;
END_FOR
(* init. Number Page *)
iPageNumber:=0;

(* QVis page 0, start page *)
iIndexPage:=0;
iPageNumber:=iPageNumber+1;
T_Visu.T_PageIndex[iIndexPage].iIndexConfigPage:=iPageNumber;
ptrConfigPage:=ADR(T_Visu.T_ConfigPage[T_Visu.T_PageIndex[iIndexPage].iIndexConfigPage]);
ptrConfigPage^.sName:='Start page';
ptrConfigPage^.wMaskBtPanelLeft:=16#0;
ptrConfigPage^.wMaskBtPanelRight:=16#0;
ptrConfigPage^.wMaskFunctionPanel:=16#0;
(* Navigation panel restriction *)
ptrConfigPage^.wMaskTouchScreenNavPanel:=16#0;
(* Active machine movement mask *)
ptrConfigPage^.wMaskActiveMachineBtPanelLeft:=16#0;
ptrConfigPage^.wMaskActiveMachineBtPanelRight:=16#0;
ptrConfigPage^.wMaskActiveMachineFunctionPanel:=16#0;
ptrConfigPage^.wMaskActiveMachineNavPanel:=16#0;
(* Button edge action *)
ptrConfigPage^.aiRTrigActionPanelRight[1]:=0;
ptrConfigPage^.aiRTrigActionPanelRight[2]:=0;
ptrConfigPage^.aiRTrigActionPanelRight[3]:=0;
ptrConfigPage^.aiRTrigActionPanelRight[4]:=0;
ptrConfigPage^.aiRTrigActionPanelRight[5]:=0;
ptrConfigPage^.aiFTrigActionPanelRight[1]:=0;
ptrConfigPage^.aiFTrigActionPanelRight[2]:=0;
ptrConfigPage^.aiFTrigActionPanelRight[3]:=0;
ptrConfigPage^.aiFTrigActionPanelRight[4]:=0;
ptrConfigPage^.aiFTrigActionPanelRight[5]:=0;
ptrConfigPage^.aiDelayActionPanelRight[1]:=0;
ptrConfigPage^.aiDelayActionPanelRight[2]:=0;
ptrConfigPage^.aiDelayActionPanelRight[3]:=0;
ptrConfigPage^.aiDelayActionPanelRight[4]:=0;
ptrConfigPage^.aiDelayActionPanelRight[5]:=0;
ptrConfigPage^.aiRTrigActionFunctionPanel[1]:=0;
ptrConfigPage^.aiRTrigActionFunctionPanel[2]:=0;
ptrConfigPage^.aiRTrigActionFunctionPanel[3]:=0;
ptrConfigPage^.aiRTrigActionFunctionPanel[4]:=0;
ptrConfigPage^.aiRTrigActionFunctionPanel[5]:=0;
ptrConfigPage^.aiRTrigActionFunctionPanel[6]:=0;
ptrConfigPage^.aiRTrigActionFunctionPanel[7]:=0;
ptrConfigPage^.aiRTrigActionFunctionPanel[8]:=0;
ptrConfigPage^.aiRTrigActionFunctionPanel[9]:=0;
ptrConfigPage^.aiRTrigActionFunctionPanel[10]:=0;
ptrConfigPage^.aiRTrigActionFunctionPanel[11]:=0;
ptrConfigPage^.aiRTrigActionFunctionPanel[12]:=0;
ptrConfigPage^.aiFTrigActionTouchScreenNavPanel[1]:=0;
ptrConfigPage^.aiFTrigActionTouchScreenNavPanel[2]:=0;
ptrConfigPage^.aiFTrigActionTouchScreenNavPanel[3]:=0;
ptrConfigPage^.aiFTrigActionTouchScreenNavPanel[4]:=0;
ptrConfigPage^.aiFTrigActionTouchScreenNavPanel[5]:=0;
ptrConfigPage^.aiFTrigActionTouchScreenNavPanel[6]:=0;
ptrConfigPage^.xMaskBtStart:=TRUE;
ptrConfigPage^.xMaskBtStop:=FALSE;

(* QVis page 1, BIOS Password StartUp *)
iIndexPage:=1;
iPageNumber:=iPageNumber+1;
T_Visu.T_PageIndex[iIndexPage].iIndexConfigPage:=iPageNumber;
ptrConfigPage:=ADR(T_Visu.T_ConfigPage[T_Visu.T_PageIndex[iIndexPage].iIndexConfigPage]);
ptrConfigPage^.sName:='BIOS Password StartUp';
ptrConfigPage^.wMaskBtPanelLeft:=16#0;
ptrConfigPage^.wMaskBtPanelRight:=16#0;
ptrConfigPage^.wMaskFunctionPanel:=16#0;
(* Navigation panel restriction *)
ptrConfigPage^.wMaskTouchScreenNavPanel:=16#0;
(* Active machine movement mask *)
ptrConfigPage^.wMaskActiveMachineBtPanelLeft:=16#0;
ptrConfigPage^.wMaskActiveMachineBtPanelRight:=16#0;
ptrConfigPage^.wMaskActiveMachineFunctionPanel:=16#0;
ptrConfigPage^.wMaskActiveMachineNavPanel:=16#0;
(* Button edge action *)
ptrConfigPage^.aiRTrigActionPanelRight[1]:=0;
ptrConfigPage^.aiRTrigActionPanelRight[2]:=0;
ptrConfigPage^.aiRTrigActionPanelRight[3]:=0;
ptrConfigPage^.aiRTrigActionPanelRight[4]:=0;
ptrConfigPage^.aiRTrigActionPanelRight[5]:=0;
ptrConfigPage^.aiFTrigActionPanelRight[1]:=0;
ptrConfigPage^.aiFTrigActionPanelRight[2]:=0;
ptrConfigPage^.aiFTrigActionPanelRight[3]:=0;
ptrConfigPage^.aiFTrigActionPanelRight[4]:=0;
ptrConfigPage^.aiFTrigActionPanelRight[5]:=0;
ptrConfigPage^.aiDelayActionPanelRight[1]:=0;
ptrConfigPage^.aiDelayActionPanelRight[2]:=0;
ptrConfigPage^.aiDelayActionPanelRight[3]:=0;
ptrConfigPage^.aiDelayActionPanelRight[4]:=0;
ptrConfigPage^.aiDelayActionPanelRight[5]:=0;
ptrConfigPage^.aiRTrigActionFunctionPanel[1]:=0;
ptrConfigPage^.aiRTrigActionFunctionPanel[2]:=0;
ptrConfigPage^.aiRTrigActionFunctionPanel[3]:=0;
ptrConfigPage^.aiRTrigActionFunctionPanel[4]:=0;
ptrConfigPage^.aiRTrigActionFunctionPanel[5]:=0;
ptrConfigPage^.aiRTrigActionFunctionPanel[6]:=0;
ptrConfigPage^.aiRTrigActionFunctionPanel[7]:=0;
ptrConfigPage^.aiRTrigActionFunctionPanel[8]:=0;
ptrConfigPage^.aiRTrigActionFunctionPanel[9]:=0;
ptrConfigPage^.aiRTrigActionFunctionPanel[10]:=0;
ptrConfigPage^.aiRTrigActionFunctionPanel[11]:=0;
ptrConfigPage^.aiRTrigActionFunctionPanel[12]:=0;
ptrConfigPage^.aiFTrigActionTouchScreenNavPanel[1]:=0;
ptrConfigPage^.aiFTrigActionTouchScreenNavPanel[2]:=0;
ptrConfigPage^.aiFTrigActionTouchScreenNavPanel[3]:=0;
ptrConfigPage^.aiFTrigActionTouchScreenNavPanel[4]:=0;
ptrConfigPage^.aiFTrigActionTouchScreenNavPanel[5]:=0;
ptrConfigPage^.aiFTrigActionTouchScreenNavPanel[6]:=0;
ptrConfigPage^.xMaskBtStart:=FALSE;
ptrConfigPage^.xMaskBtStop:=FALSE;

(* QVis page 2, BIOS Parameter StartUp *)
iIndexPage:=2;
iPageNumber:=iPageNumber+1;
T_Visu.T_PageIndex[iIndexPage].iIndexConfigPage:=iPageNumber;
ptrConfigPage:=ADR(T_Visu.T_ConfigPage[T_Visu.T_PageIndex[iIndexPage].iIndexConfigPage]);
ptrConfigPage^.sName:='BIOS Parameter StartUp';
ptrConfigPage^.wMaskBtPanelLeft:=16#0;
ptrConfigPage^.wMaskBtPanelRight:=16#200;
ptrConfigPage^.wMaskFunctionPanel:=16#0;
(* Navigation panel restriction *)
ptrConfigPage^.wMaskTouchScreenNavPanel:=16#0;
(* Active machine movement mask *)
ptrConfigPage^.wMaskActiveMachineBtPanelLeft:=16#0;
ptrConfigPage^.wMaskActiveMachineBtPanelRight:=16#200;
ptrConfigPage^.wMaskActiveMachineFunctionPanel:=16#0;
ptrConfigPage^.wMaskActiveMachineNavPanel:=16#0;
(* Button edge action *)
ptrConfigPage^.aiRTrigActionPanelRight[1]:=0;
ptrConfigPage^.aiRTrigActionPanelRight[2]:=0;
ptrConfigPage^.aiRTrigActionPanelRight[3]:=0;
ptrConfigPage^.aiRTrigActionPanelRight[4]:=0;
ptrConfigPage^.aiRTrigActionPanelRight[5]:=0;
ptrConfigPage^.aiFTrigActionPanelRight[1]:=0;
ptrConfigPage^.aiFTrigActionPanelRight[2]:=0;
ptrConfigPage^.aiFTrigActionPanelRight[3]:=0;
ptrConfigPage^.aiFTrigActionPanelRight[4]:=0;
ptrConfigPage^.aiFTrigActionPanelRight[5]:=0;
ptrConfigPage^.aiDelayActionPanelRight[1]:=0;
ptrConfigPage^.aiDelayActionPanelRight[2]:=0;
ptrConfigPage^.aiDelayActionPanelRight[3]:=0;
ptrConfigPage^.aiDelayActionPanelRight[4]:=0;
ptrConfigPage^.aiDelayActionPanelRight[5]:=0;
ptrConfigPage^.aiRTrigActionFunctionPanel[1]:=0;
ptrConfigPage^.aiRTrigActionFunctionPanel[2]:=0;
ptrConfigPage^.aiRTrigActionFunctionPanel[3]:=0;
ptrConfigPage^.aiRTrigActionFunctionPanel[4]:=0;
ptrConfigPage^.aiRTrigActionFunctionPanel[5]:=0;
ptrConfigPage^.aiRTrigActionFunctionPanel[6]:=0;
ptrConfigPage^.aiRTrigActionFunctionPanel[7]:=0;
ptrConfigPage^.aiRTrigActionFunctionPanel[8]:=0;
ptrConfigPage^.aiRTrigActionFunctionPanel[9]:=0;
ptrConfigPage^.aiRTrigActionFunctionPanel[10]:=0;
ptrConfigPage^.aiRTrigActionFunctionPanel[11]:=0;
ptrConfigPage^.aiRTrigActionFunctionPanel[12]:=0;
ptrConfigPage^.aiFTrigActionTouchScreenNavPanel[1]:=0;
ptrConfigPage^.aiFTrigActionTouchScreenNavPanel[2]:=0;
ptrConfigPage^.aiFTrigActionTouchScreenNavPanel[3]:=0;
ptrConfigPage^.aiFTrigActionTouchScreenNavPanel[4]:=0;
ptrConfigPage^.aiFTrigActionTouchScreenNavPanel[5]:=0;
ptrConfigPage^.aiFTrigActionTouchScreenNavPanel[6]:=0;
ptrConfigPage^.xMaskBtStart:=FALSE;
ptrConfigPage^.xMaskBtStop:=FALSE;

(* QVis page 10, Auto Geometry, page 1 *)
iIndexPage:=10;
iPageNumber:=iPageNumber+1;
T_Visu.T_PageIndex[iIndexPage].iIndexConfigPage:=iPageNumber;
ptrConfigPage:=ADR(T_Visu.T_ConfigPage[T_Visu.T_PageIndex[iIndexPage].iIndexConfigPage]);
ptrConfigPage^.sName:='Auto Geometry, page 1';
ptrConfigPage^.wMaskBtPanelLeft:=16#F;
ptrConfigPage^.wMaskBtPanelRight:=16#200;
(*08.07.2014: KFS	{	*)
(*ptrConfigPage^.wMaskFunctionPanel:=16#F;*)
ptrConfigPage^.wMaskFunctionPanel:=16#3F;
(*08.07.2014: KFS	}	*)
(* Navigation panel restriction *)
ptrConfigPage^.wMaskTouchScreenNavPanel:=16#3F;
(* Active machine movement mask *)
ptrConfigPage^.wMaskActiveMachineBtPanelLeft:=16#F;
ptrConfigPage^.wMaskActiveMachineBtPanelRight:=16#220;
ptrConfigPage^.wMaskActiveMachineFunctionPanel:=16#0;
ptrConfigPage^.wMaskActiveMachineNavPanel:=16#3F;
(* Button edge action *)
ptrConfigPage^.aiRTrigActionPanelRight[1]:=801;
ptrConfigPage^.aiRTrigActionPanelRight[2]:=0;
ptrConfigPage^.aiRTrigActionPanelRight[3]:=0;
ptrConfigPage^.aiRTrigActionPanelRight[4]:=0;
ptrConfigPage^.aiRTrigActionPanelRight[5]:=12;
ptrConfigPage^.aiFTrigActionPanelRight[1]:=0;
ptrConfigPage^.aiFTrigActionPanelRight[2]:=0;
ptrConfigPage^.aiFTrigActionPanelRight[3]:=0;
ptrConfigPage^.aiFTrigActionPanelRight[4]:=0;
ptrConfigPage^.aiFTrigActionPanelRight[5]:=0;
ptrConfigPage^.aiDelayActionPanelRight[1]:=0;
ptrConfigPage^.aiDelayActionPanelRight[2]:=0;
ptrConfigPage^.aiDelayActionPanelRight[3]:=0;
ptrConfigPage^.aiDelayActionPanelRight[4]:=0;
ptrConfigPage^.aiDelayActionPanelRight[5]:=0;
ptrConfigPage^.aiRTrigActionFunctionPanel[1]:=102;
ptrConfigPage^.aiRTrigActionFunctionPanel[2]:=103;
ptrConfigPage^.aiRTrigActionFunctionPanel[3]:=501;
ptrConfigPage^.aiRTrigActionFunctionPanel[4]:=106;
ptrConfigPage^.aiRTrigActionFunctionPanel[5]:=107;
ptrConfigPage^.aiRTrigActionFunctionPanel[6]:=108;
ptrConfigPage^.aiRTrigActionFunctionPanel[7]:=0;
ptrConfigPage^.aiRTrigActionFunctionPanel[8]:=0;
ptrConfigPage^.aiRTrigActionFunctionPanel[9]:=0;
ptrConfigPage^.aiRTrigActionFunctionPanel[10]:=0;
ptrConfigPage^.aiRTrigActionFunctionPanel[11]:=0;
ptrConfigPage^.aiRTrigActionFunctionPanel[12]:=0;
ptrConfigPage^.aiFTrigActionTouchScreenNavPanel[1]:=10010;
ptrConfigPage^.aiFTrigActionTouchScreenNavPanel[2]:=10020;
ptrConfigPage^.aiFTrigActionTouchScreenNavPanel[3]:=10030;
ptrConfigPage^.aiFTrigActionTouchScreenNavPanel[4]:=10040;
ptrConfigPage^.aiFTrigActionTouchScreenNavPanel[5]:=10050;
ptrConfigPage^.aiFTrigActionTouchScreenNavPanel[6]:=10060;
ptrConfigPage^.xMaskBtStart:=TRUE;
ptrConfigPage^.xMaskBtStop:=TRUE;

(* QVis page 11, Auto Geometry, page 2 *)
iIndexPage:=11;
iPageNumber:=iPageNumber+1;
T_Visu.T_PageIndex[iIndexPage].iIndexConfigPage:=iPageNumber;
ptrConfigPage:=ADR(T_Visu.T_ConfigPage[T_Visu.T_PageIndex[iIndexPage].iIndexConfigPage]);
ptrConfigPage^.sName:='Auto Geometry, page 2';
ptrConfigPage^.wMaskBtPanelLeft:=16#F;
ptrConfigPage^.wMaskBtPanelRight:=16#200;
ptrConfigPage^.wMaskFunctionPanel:=16#EF;
(* Navigation panel restriction *)
ptrConfigPage^.wMaskTouchScreenNavPanel:=16#3F;
(* Active machine movement mask *)
ptrConfigPage^.wMaskActiveMachineBtPanelLeft:=16#0;
ptrConfigPage^.wMaskActiveMachineBtPanelRight:=16#0;
ptrConfigPage^.wMaskActiveMachineFunctionPanel:=16#0;
ptrConfigPage^.wMaskActiveMachineNavPanel:=16#3F;
(* Button edge action *)
ptrConfigPage^.aiRTrigActionPanelRight[1]:=0;
ptrConfigPage^.aiRTrigActionPanelRight[2]:=0;
ptrConfigPage^.aiRTrigActionPanelRight[3]:=0;
ptrConfigPage^.aiRTrigActionPanelRight[4]:=0;
ptrConfigPage^.aiRTrigActionPanelRight[5]:=12;
ptrConfigPage^.aiFTrigActionPanelRight[1]:=0;
ptrConfigPage^.aiFTrigActionPanelRight[2]:=0;
ptrConfigPage^.aiFTrigActionPanelRight[3]:=0;
ptrConfigPage^.aiFTrigActionPanelRight[4]:=0;
ptrConfigPage^.aiFTrigActionPanelRight[5]:=0;
ptrConfigPage^.aiDelayActionPanelRight[1]:=0;
ptrConfigPage^.aiDelayActionPanelRight[2]:=0;
ptrConfigPage^.aiDelayActionPanelRight[3]:=0;
ptrConfigPage^.aiDelayActionPanelRight[4]:=0;
ptrConfigPage^.aiDelayActionPanelRight[5]:=0;
ptrConfigPage^.aiRTrigActionFunctionPanel[1]:=110;
ptrConfigPage^.aiRTrigActionFunctionPanel[2]:=111;
ptrConfigPage^.aiRTrigActionFunctionPanel[3]:=114;
ptrConfigPage^.aiRTrigActionFunctionPanel[4]:=115;
ptrConfigPage^.aiRTrigActionFunctionPanel[5]:=0;
ptrConfigPage^.aiRTrigActionFunctionPanel[6]:=116;
ptrConfigPage^.aiRTrigActionFunctionPanel[7]:=112;
ptrConfigPage^.aiRTrigActionFunctionPanel[8]:=113;
ptrConfigPage^.aiRTrigActionFunctionPanel[9]:=0;
ptrConfigPage^.aiRTrigActionFunctionPanel[10]:=0;
ptrConfigPage^.aiRTrigActionFunctionPanel[11]:=0;
ptrConfigPage^.aiRTrigActionFunctionPanel[12]:=0;
ptrConfigPage^.aiFTrigActionTouchScreenNavPanel[1]:=10010;
ptrConfigPage^.aiFTrigActionTouchScreenNavPanel[2]:=10020;
ptrConfigPage^.aiFTrigActionTouchScreenNavPanel[3]:=10030;
ptrConfigPage^.aiFTrigActionTouchScreenNavPanel[4]:=10040;
ptrConfigPage^.aiFTrigActionTouchScreenNavPanel[5]:=10050;
ptrConfigPage^.aiFTrigActionTouchScreenNavPanel[6]:=10060;
ptrConfigPage^.xMaskBtStart:=TRUE;
ptrConfigPage^.xMaskBtStop:=TRUE;

(* QVis page 20, Auto Groove, page 1 *)
iIndexPage:=20;
iPageNumber:=iPageNumber+1;
T_Visu.T_PageIndex[iIndexPage].iIndexConfigPage:=iPageNumber;
ptrConfigPage:=ADR(T_Visu.T_ConfigPage[T_Visu.T_PageIndex[iIndexPage].iIndexConfigPage]);
ptrConfigPage^.sName:='Auto Groove, page 1';
ptrConfigPage^.wMaskBtPanelLeft:=16#F;
ptrConfigPage^.wMaskBtPanelRight:=16#200;
ptrConfigPage^.wMaskFunctionPanel:=16#3F;
(* Navigation panel restriction *)
ptrConfigPage^.wMaskTouchScreenNavPanel:=16#3F;
(* Active machine movement mask *)
ptrConfigPage^.wMaskActiveMachineBtPanelLeft:=16#F;
ptrConfigPage^.wMaskActiveMachineBtPanelRight:=16#200;
ptrConfigPage^.wMaskActiveMachineFunctionPanel:=16#0;
ptrConfigPage^.wMaskActiveMachineNavPanel:=16#3F;
(* Button edge action *)
ptrConfigPage^.aiRTrigActionPanelRight[1]:=0;
ptrConfigPage^.aiRTrigActionPanelRight[2]:=0;
ptrConfigPage^.aiRTrigActionPanelRight[3]:=0;
ptrConfigPage^.aiRTrigActionPanelRight[4]:=0;
ptrConfigPage^.aiRTrigActionPanelRight[5]:=12;
ptrConfigPage^.aiFTrigActionPanelRight[1]:=0;
ptrConfigPage^.aiFTrigActionPanelRight[2]:=0;
ptrConfigPage^.aiFTrigActionPanelRight[3]:=0;
ptrConfigPage^.aiFTrigActionPanelRight[4]:=0;
ptrConfigPage^.aiFTrigActionPanelRight[5]:=0;
ptrConfigPage^.aiDelayActionPanelRight[1]:=0;
ptrConfigPage^.aiDelayActionPanelRight[2]:=0;
ptrConfigPage^.aiDelayActionPanelRight[3]:=0;
ptrConfigPage^.aiDelayActionPanelRight[4]:=0;
ptrConfigPage^.aiDelayActionPanelRight[5]:=0;
ptrConfigPage^.aiRTrigActionFunctionPanel[1]:=102;
ptrConfigPage^.aiRTrigActionFunctionPanel[2]:=103;
ptrConfigPage^.aiRTrigActionFunctionPanel[3]:=501;
ptrConfigPage^.aiRTrigActionFunctionPanel[4]:=105;
ptrConfigPage^.aiRTrigActionFunctionPanel[5]:=107;
ptrConfigPage^.aiRTrigActionFunctionPanel[6]:=104;
ptrConfigPage^.aiRTrigActionFunctionPanel[7]:=0;
ptrConfigPage^.aiRTrigActionFunctionPanel[8]:=0;
ptrConfigPage^.aiRTrigActionFunctionPanel[9]:=0;
ptrConfigPage^.aiRTrigActionFunctionPanel[10]:=0;
ptrConfigPage^.aiRTrigActionFunctionPanel[11]:=0;
ptrConfigPage^.aiRTrigActionFunctionPanel[12]:=0;
ptrConfigPage^.aiFTrigActionTouchScreenNavPanel[1]:=10010;
ptrConfigPage^.aiFTrigActionTouchScreenNavPanel[2]:=10020;
ptrConfigPage^.aiFTrigActionTouchScreenNavPanel[3]:=10030;
ptrConfigPage^.aiFTrigActionTouchScreenNavPanel[4]:=10040;
ptrConfigPage^.aiFTrigActionTouchScreenNavPanel[5]:=10050;
ptrConfigPage^.aiFTrigActionTouchScreenNavPanel[6]:=10060;
ptrConfigPage^.xMaskBtStart:=TRUE;
ptrConfigPage^.xMaskBtStop:=TRUE;

(* QVis page 21, Auto Groove, page 2 *)
iIndexPage:=21;
iPageNumber:=iPageNumber+1;
T_Visu.T_PageIndex[iIndexPage].iIndexConfigPage:=iPageNumber;
ptrConfigPage:=ADR(T_Visu.T_ConfigPage[T_Visu.T_PageIndex[iIndexPage].iIndexConfigPage]);
ptrConfigPage^.sName:='Auto Groove, page 2';
ptrConfigPage^.wMaskBtPanelLeft:=16#F;
ptrConfigPage^.wMaskBtPanelRight:=16#200;
ptrConfigPage^.wMaskFunctionPanel:=16#EF;
(* Navigation panel restriction *)
ptrConfigPage^.wMaskTouchScreenNavPanel:=16#3F;
(* Active machine movement mask *)
ptrConfigPage^.wMaskActiveMachineBtPanelLeft:=16#0;
ptrConfigPage^.wMaskActiveMachineBtPanelRight:=16#0;
ptrConfigPage^.wMaskActiveMachineFunctionPanel:=16#0;
ptrConfigPage^.wMaskActiveMachineNavPanel:=16#3F;
(* Button edge action *)
ptrConfigPage^.aiRTrigActionPanelRight[1]:=0;
ptrConfigPage^.aiRTrigActionPanelRight[2]:=0;
ptrConfigPage^.aiRTrigActionPanelRight[3]:=0;
ptrConfigPage^.aiRTrigActionPanelRight[4]:=0;
ptrConfigPage^.aiRTrigActionPanelRight[5]:=12;
ptrConfigPage^.aiFTrigActionPanelRight[1]:=0;
ptrConfigPage^.aiFTrigActionPanelRight[2]:=0;
ptrConfigPage^.aiFTrigActionPanelRight[3]:=0;
ptrConfigPage^.aiFTrigActionPanelRight[4]:=0;
ptrConfigPage^.aiFTrigActionPanelRight[5]:=0;
ptrConfigPage^.aiDelayActionPanelRight[1]:=0;
ptrConfigPage^.aiDelayActionPanelRight[2]:=0;
ptrConfigPage^.aiDelayActionPanelRight[3]:=0;
ptrConfigPage^.aiDelayActionPanelRight[4]:=0;
ptrConfigPage^.aiDelayActionPanelRight[5]:=0;
ptrConfigPage^.aiRTrigActionFunctionPanel[1]:=110;
ptrConfigPage^.aiRTrigActionFunctionPanel[2]:=111;
ptrConfigPage^.aiRTrigActionFunctionPanel[3]:=114;
ptrConfigPage^.aiRTrigActionFunctionPanel[4]:=115;
ptrConfigPage^.aiRTrigActionFunctionPanel[5]:=0;
ptrConfigPage^.aiRTrigActionFunctionPanel[6]:=116;
ptrConfigPage^.aiRTrigActionFunctionPanel[7]:=112;
ptrConfigPage^.aiRTrigActionFunctionPanel[8]:=113;
ptrConfigPage^.aiRTrigActionFunctionPanel[9]:=0;
ptrConfigPage^.aiRTrigActionFunctionPanel[10]:=0;
ptrConfigPage^.aiRTrigActionFunctionPanel[11]:=0;
ptrConfigPage^.aiRTrigActionFunctionPanel[12]:=0;
ptrConfigPage^.aiFTrigActionTouchScreenNavPanel[1]:=10010;
ptrConfigPage^.aiFTrigActionTouchScreenNavPanel[2]:=10020;
ptrConfigPage^.aiFTrigActionTouchScreenNavPanel[3]:=10030;
ptrConfigPage^.aiFTrigActionTouchScreenNavPanel[4]:=10040;
ptrConfigPage^.aiFTrigActionTouchScreenNavPanel[5]:=10050;
ptrConfigPage^.aiFTrigActionTouchScreenNavPanel[6]:=10060;
ptrConfigPage^.xMaskBtStart:=TRUE;
ptrConfigPage^.xMaskBtStop:=TRUE;

(* QVis page 30, Reference *)
iIndexPage:=30;
iPageNumber:=iPageNumber+1;
T_Visu.T_PageIndex[iIndexPage].iIndexConfigPage:=iPageNumber;
ptrConfigPage:=ADR(T_Visu.T_ConfigPage[T_Visu.T_PageIndex[iIndexPage].iIndexConfigPage]);
ptrConfigPage^.sName:='Reference';
ptrConfigPage^.wMaskBtPanelLeft:=16#F;
ptrConfigPage^.wMaskBtPanelRight:=16#1E0;
ptrConfigPage^.wMaskFunctionPanel:=16#D;
(* Navigation panel restriction *)
ptrConfigPage^.wMaskTouchScreenNavPanel:=16#3F;
(* Active machine movement mask *)
ptrConfigPage^.wMaskActiveMachineBtPanelLeft:=16#F;
ptrConfigPage^.wMaskActiveMachineBtPanelRight:=16#60;
ptrConfigPage^.wMaskActiveMachineFunctionPanel:=16#0;
ptrConfigPage^.wMaskActiveMachineNavPanel:=16#3F;
(* Button edge action *)
ptrConfigPage^.aiRTrigActionPanelRight[1]:=312;
ptrConfigPage^.aiRTrigActionPanelRight[2]:=310;
ptrConfigPage^.aiRTrigActionPanelRight[3]:=316;
ptrConfigPage^.aiRTrigActionPanelRight[4]:=314;
ptrConfigPage^.aiRTrigActionPanelRight[5]:=0;
ptrConfigPage^.aiFTrigActionPanelRight[1]:=0;
ptrConfigPage^.aiFTrigActionPanelRight[2]:=0;
ptrConfigPage^.aiFTrigActionPanelRight[3]:=301;
ptrConfigPage^.aiFTrigActionPanelRight[4]:=301;
ptrConfigPage^.aiFTrigActionPanelRight[5]:=0;
ptrConfigPage^.aiDelayActionPanelRight[1]:=0;
ptrConfigPage^.aiDelayActionPanelRight[2]:=0;
ptrConfigPage^.aiDelayActionPanelRight[3]:=0;
ptrConfigPage^.aiDelayActionPanelRight[4]:=0;
ptrConfigPage^.aiDelayActionPanelRight[5]:=0;
ptrConfigPage^.aiRTrigActionFunctionPanel[1]:=320;
ptrConfigPage^.aiRTrigActionFunctionPanel[2]:=0;
ptrConfigPage^.aiRTrigActionFunctionPanel[3]:=501;
ptrConfigPage^.aiRTrigActionFunctionPanel[4]:=106;
ptrConfigPage^.aiRTrigActionFunctionPanel[5]:=0;
ptrConfigPage^.aiRTrigActionFunctionPanel[6]:=0;
ptrConfigPage^.aiRTrigActionFunctionPanel[7]:=0;
ptrConfigPage^.aiRTrigActionFunctionPanel[8]:=0;
ptrConfigPage^.aiRTrigActionFunctionPanel[9]:=0;
ptrConfigPage^.aiRTrigActionFunctionPanel[10]:=0;
ptrConfigPage^.aiRTrigActionFunctionPanel[11]:=0;
ptrConfigPage^.aiRTrigActionFunctionPanel[12]:=0;
ptrConfigPage^.aiFTrigActionTouchScreenNavPanel[1]:=10010;
ptrConfigPage^.aiFTrigActionTouchScreenNavPanel[2]:=10020;
ptrConfigPage^.aiFTrigActionTouchScreenNavPanel[3]:=10030;
ptrConfigPage^.aiFTrigActionTouchScreenNavPanel[4]:=10040;
ptrConfigPage^.aiFTrigActionTouchScreenNavPanel[5]:=10050;
ptrConfigPage^.aiFTrigActionTouchScreenNavPanel[6]:=10060;
ptrConfigPage^.xMaskBtStart:=TRUE;
ptrConfigPage^.xMaskBtStop:=TRUE;

(* QVis page 40, Setup --> change user level *)
iIndexPage:=40;
iPageNumber:=iPageNumber+1;
T_Visu.T_PageIndex[iIndexPage].iIndexConfigPage:=iPageNumber;
ptrConfigPage:=ADR(T_Visu.T_ConfigPage[T_Visu.T_PageIndex[iIndexPage].iIndexConfigPage]);
ptrConfigPage^.sName:='Setup --> change user level';
ptrConfigPage^.wMaskBtPanelLeft:=16#F;
ptrConfigPage^.wMaskBtPanelRight:=16#200;
ptrConfigPage^.wMaskFunctionPanel:=16#0;
(* Navigation panel restriction *)
ptrConfigPage^.wMaskTouchScreenNavPanel:=16#3F;
(* Active machine movement mask *)
ptrConfigPage^.wMaskActiveMachineBtPanelLeft:=16#0;
ptrConfigPage^.wMaskActiveMachineBtPanelRight:=16#200;
ptrConfigPage^.wMaskActiveMachineFunctionPanel:=16#0;
ptrConfigPage^.wMaskActiveMachineNavPanel:=16#3F;
(* Button edge action *)
ptrConfigPage^.aiRTrigActionPanelRight[1]:=0;
ptrConfigPage^.aiRTrigActionPanelRight[2]:=0;
ptrConfigPage^.aiRTrigActionPanelRight[3]:=0;
ptrConfigPage^.aiRTrigActionPanelRight[4]:=0;
ptrConfigPage^.aiRTrigActionPanelRight[5]:=12;
ptrConfigPage^.aiFTrigActionPanelRight[1]:=0;
ptrConfigPage^.aiFTrigActionPanelRight[2]:=0;
ptrConfigPage^.aiFTrigActionPanelRight[3]:=0;
ptrConfigPage^.aiFTrigActionPanelRight[4]:=0;
ptrConfigPage^.aiFTrigActionPanelRight[5]:=0;
ptrConfigPage^.aiDelayActionPanelRight[1]:=0;
ptrConfigPage^.aiDelayActionPanelRight[2]:=0;
ptrConfigPage^.aiDelayActionPanelRight[3]:=0;
ptrConfigPage^.aiDelayActionPanelRight[4]:=0;
ptrConfigPage^.aiDelayActionPanelRight[5]:=0;
ptrConfigPage^.aiRTrigActionFunctionPanel[1]:=0;
ptrConfigPage^.aiRTrigActionFunctionPanel[2]:=0;
ptrConfigPage^.aiRTrigActionFunctionPanel[3]:=0;
ptrConfigPage^.aiRTrigActionFunctionPanel[4]:=0;
ptrConfigPage^.aiRTrigActionFunctionPanel[5]:=0;
ptrConfigPage^.aiRTrigActionFunctionPanel[6]:=0;
ptrConfigPage^.aiRTrigActionFunctionPanel[7]:=0;
ptrConfigPage^.aiRTrigActionFunctionPanel[8]:=0;
ptrConfigPage^.aiRTrigActionFunctionPanel[9]:=0;
ptrConfigPage^.aiRTrigActionFunctionPanel[10]:=0;
ptrConfigPage^.aiRTrigActionFunctionPanel[11]:=0;
ptrConfigPage^.aiRTrigActionFunctionPanel[12]:=0;
ptrConfigPage^.aiFTrigActionTouchScreenNavPanel[1]:=10010;
ptrConfigPage^.aiFTrigActionTouchScreenNavPanel[2]:=10020;
ptrConfigPage^.aiFTrigActionTouchScreenNavPanel[3]:=10030;
ptrConfigPage^.aiFTrigActionTouchScreenNavPanel[4]:=10040;
ptrConfigPage^.aiFTrigActionTouchScreenNavPanel[5]:=10050;
ptrConfigPage^.aiFTrigActionTouchScreenNavPanel[6]:=10060;
ptrConfigPage^.xMaskBtStart:=FALSE;
ptrConfigPage^.xMaskBtStop:=TRUE;

(* QVis page 41, Setup --> change language *)
iIndexPage:=41;
iPageNumber:=iPageNumber+1;
T_Visu.T_PageIndex[iIndexPage].iIndexConfigPage:=iPageNumber;
ptrConfigPage:=ADR(T_Visu.T_ConfigPage[T_Visu.T_PageIndex[iIndexPage].iIndexConfigPage]);
ptrConfigPage^.sName:='Setup --> change language';
ptrConfigPage^.wMaskBtPanelLeft:=16#F;
ptrConfigPage^.wMaskBtPanelRight:=16#200;
ptrConfigPage^.wMaskFunctionPanel:=16#0;
(* Navigation panel restriction *)
ptrConfigPage^.wMaskTouchScreenNavPanel:=16#3F;
(* Active machine movement mask *)
ptrConfigPage^.wMaskActiveMachineBtPanelLeft:=16#0;
ptrConfigPage^.wMaskActiveMachineBtPanelRight:=16#200;
ptrConfigPage^.wMaskActiveMachineFunctionPanel:=16#0;
ptrConfigPage^.wMaskActiveMachineNavPanel:=16#3F;
(* Button edge action *)
ptrConfigPage^.aiRTrigActionPanelRight[1]:=0;
ptrConfigPage^.aiRTrigActionPanelRight[2]:=0;
ptrConfigPage^.aiRTrigActionPanelRight[3]:=0;
ptrConfigPage^.aiRTrigActionPanelRight[4]:=0;
ptrConfigPage^.aiRTrigActionPanelRight[5]:=12;
ptrConfigPage^.aiFTrigActionPanelRight[1]:=0;
ptrConfigPage^.aiFTrigActionPanelRight[2]:=0;
ptrConfigPage^.aiFTrigActionPanelRight[3]:=0;
ptrConfigPage^.aiFTrigActionPanelRight[4]:=0;
ptrConfigPage^.aiFTrigActionPanelRight[5]:=0;
ptrConfigPage^.aiDelayActionPanelRight[1]:=0;
ptrConfigPage^.aiDelayActionPanelRight[2]:=0;
ptrConfigPage^.aiDelayActionPanelRight[3]:=0;
ptrConfigPage^.aiDelayActionPanelRight[4]:=0;
ptrConfigPage^.aiDelayActionPanelRight[5]:=0;
ptrConfigPage^.aiRTrigActionFunctionPanel[1]:=0;
ptrConfigPage^.aiRTrigActionFunctionPanel[2]:=0;
ptrConfigPage^.aiRTrigActionFunctionPanel[3]:=0;
ptrConfigPage^.aiRTrigActionFunctionPanel[4]:=0;
ptrConfigPage^.aiRTrigActionFunctionPanel[5]:=0;
ptrConfigPage^.aiRTrigActionFunctionPanel[6]:=0;
ptrConfigPage^.aiRTrigActionFunctionPanel[7]:=0;
ptrConfigPage^.aiRTrigActionFunctionPanel[8]:=0;
ptrConfigPage^.aiRTrigActionFunctionPanel[9]:=0;
ptrConfigPage^.aiRTrigActionFunctionPanel[10]:=0;
ptrConfigPage^.aiRTrigActionFunctionPanel[11]:=0;
ptrConfigPage^.aiRTrigActionFunctionPanel[12]:=0;
ptrConfigPage^.aiFTrigActionTouchScreenNavPanel[1]:=10010;
ptrConfigPage^.aiFTrigActionTouchScreenNavPanel[2]:=10020;
ptrConfigPage^.aiFTrigActionTouchScreenNavPanel[3]:=10030;
ptrConfigPage^.aiFTrigActionTouchScreenNavPanel[4]:=10040;
ptrConfigPage^.aiFTrigActionTouchScreenNavPanel[5]:=10050;
ptrConfigPage^.aiFTrigActionTouchScreenNavPanel[6]:=10060;
ptrConfigPage^.xMaskBtStart:=FALSE;
ptrConfigPage^.xMaskBtStop:=TRUE;

(* QVis page 50, Axis informations *)
iIndexPage:=50;
iPageNumber:=iPageNumber+1;
T_Visu.T_PageIndex[iIndexPage].iIndexConfigPage:=iPageNumber;
ptrConfigPage:=ADR(T_Visu.T_ConfigPage[T_Visu.T_PageIndex[iIndexPage].iIndexConfigPage]);
ptrConfigPage^.sName:='Axis informations';
ptrConfigPage^.wMaskBtPanelLeft:=16#F;
ptrConfigPage^.wMaskBtPanelRight:=16#200;
ptrConfigPage^.wMaskFunctionPanel:=16#0;
(* Navigation panel restriction *)
ptrConfigPage^.wMaskTouchScreenNavPanel:=16#3F;
(* Active machine movement mask *)
ptrConfigPage^.wMaskActiveMachineBtPanelLeft:=16#0;
ptrConfigPage^.wMaskActiveMachineBtPanelRight:=16#200;
ptrConfigPage^.wMaskActiveMachineFunctionPanel:=16#0;
ptrConfigPage^.wMaskActiveMachineNavPanel:=16#3F;
(* Button edge action *)
ptrConfigPage^.aiRTrigActionPanelRight[1]:=0;
ptrConfigPage^.aiRTrigActionPanelRight[2]:=0;
ptrConfigPage^.aiRTrigActionPanelRight[3]:=0;
ptrConfigPage^.aiRTrigActionPanelRight[4]:=0;
ptrConfigPage^.aiRTrigActionPanelRight[5]:=12;
ptrConfigPage^.aiFTrigActionPanelRight[1]:=0;
ptrConfigPage^.aiFTrigActionPanelRight[2]:=0;
ptrConfigPage^.aiFTrigActionPanelRight[3]:=0;
ptrConfigPage^.aiFTrigActionPanelRight[4]:=0;
ptrConfigPage^.aiFTrigActionPanelRight[5]:=0;
ptrConfigPage^.aiDelayActionPanelRight[1]:=0;
ptrConfigPage^.aiDelayActionPanelRight[2]:=0;
ptrConfigPage^.aiDelayActionPanelRight[3]:=0;
ptrConfigPage^.aiDelayActionPanelRight[4]:=0;
ptrConfigPage^.aiDelayActionPanelRight[5]:=0;
ptrConfigPage^.aiRTrigActionFunctionPanel[1]:=0;
ptrConfigPage^.aiRTrigActionFunctionPanel[2]:=0;
ptrConfigPage^.aiRTrigActionFunctionPanel[3]:=0;
ptrConfigPage^.aiRTrigActionFunctionPanel[4]:=0;
ptrConfigPage^.aiRTrigActionFunctionPanel[5]:=0;
ptrConfigPage^.aiRTrigActionFunctionPanel[6]:=0;
ptrConfigPage^.aiRTrigActionFunctionPanel[7]:=0;
ptrConfigPage^.aiRTrigActionFunctionPanel[8]:=0;
ptrConfigPage^.aiRTrigActionFunctionPanel[9]:=0;
ptrConfigPage^.aiRTrigActionFunctionPanel[10]:=0;
ptrConfigPage^.aiRTrigActionFunctionPanel[11]:=0;
ptrConfigPage^.aiRTrigActionFunctionPanel[12]:=0;
ptrConfigPage^.aiFTrigActionTouchScreenNavPanel[1]:=10010;
ptrConfigPage^.aiFTrigActionTouchScreenNavPanel[2]:=10020;
ptrConfigPage^.aiFTrigActionTouchScreenNavPanel[3]:=10030;
ptrConfigPage^.aiFTrigActionTouchScreenNavPanel[4]:=10040;
ptrConfigPage^.aiFTrigActionTouchScreenNavPanel[5]:=10050;
ptrConfigPage^.aiFTrigActionTouchScreenNavPanel[6]:=10060;
ptrConfigPage^.xMaskBtStart:=FALSE;
ptrConfigPage^.xMaskBtStop:=TRUE;

(* QVis page 51, System informations *)
iIndexPage:=51;
iPageNumber:=iPageNumber+1;
T_Visu.T_PageIndex[iIndexPage].iIndexConfigPage:=iPageNumber;
ptrConfigPage:=ADR(T_Visu.T_ConfigPage[T_Visu.T_PageIndex[iIndexPage].iIndexConfigPage]);
ptrConfigPage^.sName:='System informations';
ptrConfigPage^.wMaskBtPanelLeft:=16#F;
ptrConfigPage^.wMaskBtPanelRight:=16#200;
ptrConfigPage^.wMaskFunctionPanel:=16#0;
(* Navigation panel restriction *)
ptrConfigPage^.wMaskTouchScreenNavPanel:=16#3F;
(* Active machine movement mask *)
ptrConfigPage^.wMaskActiveMachineBtPanelLeft:=16#0;
ptrConfigPage^.wMaskActiveMachineBtPanelRight:=16#200;
ptrConfigPage^.wMaskActiveMachineFunctionPanel:=16#0;
ptrConfigPage^.wMaskActiveMachineNavPanel:=16#3F;
(* Button edge action *)
ptrConfigPage^.aiRTrigActionPanelRight[1]:=0;
ptrConfigPage^.aiRTrigActionPanelRight[2]:=0;
ptrConfigPage^.aiRTrigActionPanelRight[3]:=0;
ptrConfigPage^.aiRTrigActionPanelRight[4]:=0;
ptrConfigPage^.aiRTrigActionPanelRight[5]:=12;
ptrConfigPage^.aiFTrigActionPanelRight[1]:=0;
ptrConfigPage^.aiFTrigActionPanelRight[2]:=0;
ptrConfigPage^.aiFTrigActionPanelRight[3]:=0;
ptrConfigPage^.aiFTrigActionPanelRight[4]:=0;
ptrConfigPage^.aiFTrigActionPanelRight[5]:=0;
ptrConfigPage^.aiDelayActionPanelRight[1]:=0;
ptrConfigPage^.aiDelayActionPanelRight[2]:=0;
ptrConfigPage^.aiDelayActionPanelRight[3]:=0;
ptrConfigPage^.aiDelayActionPanelRight[4]:=0;
ptrConfigPage^.aiDelayActionPanelRight[5]:=0;
ptrConfigPage^.aiRTrigActionFunctionPanel[1]:=0;
ptrConfigPage^.aiRTrigActionFunctionPanel[2]:=0;
ptrConfigPage^.aiRTrigActionFunctionPanel[3]:=0;
ptrConfigPage^.aiRTrigActionFunctionPanel[4]:=0;
ptrConfigPage^.aiRTrigActionFunctionPanel[5]:=0;
ptrConfigPage^.aiRTrigActionFunctionPanel[6]:=0;
ptrConfigPage^.aiRTrigActionFunctionPanel[7]:=0;
ptrConfigPage^.aiRTrigActionFunctionPanel[8]:=0;
ptrConfigPage^.aiRTrigActionFunctionPanel[9]:=0;
ptrConfigPage^.aiRTrigActionFunctionPanel[10]:=0;
ptrConfigPage^.aiRTrigActionFunctionPanel[11]:=0;
ptrConfigPage^.aiRTrigActionFunctionPanel[12]:=0;
ptrConfigPage^.aiFTrigActionTouchScreenNavPanel[1]:=10010;
ptrConfigPage^.aiFTrigActionTouchScreenNavPanel[2]:=10020;
ptrConfigPage^.aiFTrigActionTouchScreenNavPanel[3]:=10030;
ptrConfigPage^.aiFTrigActionTouchScreenNavPanel[4]:=10040;
ptrConfigPage^.aiFTrigActionTouchScreenNavPanel[5]:=10050;
ptrConfigPage^.aiFTrigActionTouchScreenNavPanel[6]:=10060;
ptrConfigPage^.xMaskBtStart:=FALSE;
ptrConfigPage^.xMaskBtStop:=TRUE;

(* QVis page 60, Error List *)
iIndexPage:=60;
iPageNumber:=iPageNumber+1;
T_Visu.T_PageIndex[iIndexPage].iIndexConfigPage:=iPageNumber;
ptrConfigPage:=ADR(T_Visu.T_ConfigPage[T_Visu.T_PageIndex[iIndexPage].iIndexConfigPage]);
ptrConfigPage^.sName:='Error List';
ptrConfigPage^.wMaskBtPanelLeft:=16#F;
ptrConfigPage^.wMaskBtPanelRight:=16#60;
ptrConfigPage^.wMaskFunctionPanel:=16#0;
(* Navigation panel restriction *)
ptrConfigPage^.wMaskTouchScreenNavPanel:=16#3F;
(* Active machine movement mask *)
ptrConfigPage^.wMaskActiveMachineBtPanelLeft:=16#0;
ptrConfigPage^.wMaskActiveMachineBtPanelRight:=16#60;
ptrConfigPage^.wMaskActiveMachineFunctionPanel:=16#0;
ptrConfigPage^.wMaskActiveMachineNavPanel:=16#3F;
(* Button edge action *)
ptrConfigPage^.aiRTrigActionPanelRight[1]:=99;
ptrConfigPage^.aiRTrigActionPanelRight[2]:=20;
ptrConfigPage^.aiRTrigActionPanelRight[3]:=0;
ptrConfigPage^.aiRTrigActionPanelRight[4]:=0;
ptrConfigPage^.aiRTrigActionPanelRight[5]:=0;
ptrConfigPage^.aiFTrigActionPanelRight[1]:=0;
ptrConfigPage^.aiFTrigActionPanelRight[2]:=0;
ptrConfigPage^.aiFTrigActionPanelRight[3]:=0;
ptrConfigPage^.aiFTrigActionPanelRight[4]:=0;
ptrConfigPage^.aiFTrigActionPanelRight[5]:=0;
ptrConfigPage^.aiDelayActionPanelRight[1]:=0;
ptrConfigPage^.aiDelayActionPanelRight[2]:=0;
ptrConfigPage^.aiDelayActionPanelRight[3]:=0;
ptrConfigPage^.aiDelayActionPanelRight[4]:=0;
ptrConfigPage^.aiDelayActionPanelRight[5]:=0;
ptrConfigPage^.aiRTrigActionFunctionPanel[1]:=0;
ptrConfigPage^.aiRTrigActionFunctionPanel[2]:=0;
ptrConfigPage^.aiRTrigActionFunctionPanel[3]:=0;
ptrConfigPage^.aiRTrigActionFunctionPanel[4]:=0;
ptrConfigPage^.aiRTrigActionFunctionPanel[5]:=0;
ptrConfigPage^.aiRTrigActionFunctionPanel[6]:=0;
ptrConfigPage^.aiRTrigActionFunctionPanel[7]:=0;
ptrConfigPage^.aiRTrigActionFunctionPanel[8]:=0;
ptrConfigPage^.aiRTrigActionFunctionPanel[9]:=0;
ptrConfigPage^.aiRTrigActionFunctionPanel[10]:=0;
ptrConfigPage^.aiRTrigActionFunctionPanel[11]:=0;
ptrConfigPage^.aiRTrigActionFunctionPanel[12]:=0;
ptrConfigPage^.aiFTrigActionTouchScreenNavPanel[1]:=10010;
ptrConfigPage^.aiFTrigActionTouchScreenNavPanel[2]:=10020;
ptrConfigPage^.aiFTrigActionTouchScreenNavPanel[3]:=10030;
ptrConfigPage^.aiFTrigActionTouchScreenNavPanel[4]:=10040;
ptrConfigPage^.aiFTrigActionTouchScreenNavPanel[5]:=10050;
ptrConfigPage^.aiFTrigActionTouchScreenNavPanel[6]:=10060;
ptrConfigPage^.xMaskBtStart:=FALSE;
ptrConfigPage^.xMaskBtStop:=TRUE;

(* QVis page 110, Tool Calibration *)
iIndexPage:=110;
iPageNumber:=iPageNumber+1;
T_Visu.T_PageIndex[iIndexPage].iIndexConfigPage:=iPageNumber;
ptrConfigPage:=ADR(T_Visu.T_ConfigPage[T_Visu.T_PageIndex[iIndexPage].iIndexConfigPage]);
ptrConfigPage^.sName:='Tool Calibration';
ptrConfigPage^.wMaskBtPanelLeft:=16#1F;
ptrConfigPage^.wMaskBtPanelRight:=16#0;
ptrConfigPage^.wMaskFunctionPanel:=16#3F;
(* Navigation panel restriction *)
ptrConfigPage^.wMaskTouchScreenNavPanel:=16#3F;
(* Active machine movement mask *)
ptrConfigPage^.wMaskActiveMachineBtPanelLeft:=16#F;
ptrConfigPage^.wMaskActiveMachineBtPanelRight:=16#0;
ptrConfigPage^.wMaskActiveMachineFunctionPanel:=16#0;
ptrConfigPage^.wMaskActiveMachineNavPanel:=16#3F;
(* Button edge action *)
ptrConfigPage^.aiRTrigActionPanelRight[1]:=0;
ptrConfigPage^.aiRTrigActionPanelRight[2]:=0;
ptrConfigPage^.aiRTrigActionPanelRight[3]:=0;
ptrConfigPage^.aiRTrigActionPanelRight[4]:=0;
ptrConfigPage^.aiRTrigActionPanelRight[5]:=0;
ptrConfigPage^.aiFTrigActionPanelRight[1]:=0;
ptrConfigPage^.aiFTrigActionPanelRight[2]:=0;
ptrConfigPage^.aiFTrigActionPanelRight[3]:=0;
ptrConfigPage^.aiFTrigActionPanelRight[4]:=0;
ptrConfigPage^.aiFTrigActionPanelRight[5]:=0;
ptrConfigPage^.aiDelayActionPanelRight[1]:=0;
ptrConfigPage^.aiDelayActionPanelRight[2]:=0;
ptrConfigPage^.aiDelayActionPanelRight[3]:=0;
ptrConfigPage^.aiDelayActionPanelRight[4]:=0;
ptrConfigPage^.aiDelayActionPanelRight[5]:=0;
ptrConfigPage^.aiRTrigActionFunctionPanel[1]:=102;
ptrConfigPage^.aiRTrigActionFunctionPanel[2]:=103;
ptrConfigPage^.aiRTrigActionFunctionPanel[3]:=501;
ptrConfigPage^.aiRTrigActionFunctionPanel[4]:=132;
ptrConfigPage^.aiRTrigActionFunctionPanel[5]:=105;
ptrConfigPage^.aiRTrigActionFunctionPanel[6]:=101;
ptrConfigPage^.aiRTrigActionFunctionPanel[7]:=0;
ptrConfigPage^.aiRTrigActionFunctionPanel[8]:=0;
ptrConfigPage^.aiRTrigActionFunctionPanel[9]:=0;
ptrConfigPage^.aiRTrigActionFunctionPanel[10]:=0;
ptrConfigPage^.aiRTrigActionFunctionPanel[11]:=0;
ptrConfigPage^.aiRTrigActionFunctionPanel[12]:=0;
ptrConfigPage^.aiFTrigActionTouchScreenNavPanel[1]:=10110;
ptrConfigPage^.aiFTrigActionTouchScreenNavPanel[2]:=10120;
ptrConfigPage^.aiFTrigActionTouchScreenNavPanel[3]:=10130;
ptrConfigPage^.aiFTrigActionTouchScreenNavPanel[4]:=10140;
ptrConfigPage^.aiFTrigActionTouchScreenNavPanel[5]:=10150;
ptrConfigPage^.aiFTrigActionTouchScreenNavPanel[6]:=10160;
ptrConfigPage^.xMaskBtStart:=TRUE;
ptrConfigPage^.xMaskBtStop:=TRUE;

(* QVis page 120, Tool Geometry *)
iIndexPage:=120;
iPageNumber:=iPageNumber+1;
T_Visu.T_PageIndex[iIndexPage].iIndexConfigPage:=iPageNumber;
ptrConfigPage:=ADR(T_Visu.T_ConfigPage[T_Visu.T_PageIndex[iIndexPage].iIndexConfigPage]);
ptrConfigPage^.sName:='Tool Geometry';
ptrConfigPage^.wMaskBtPanelLeft:=16#1F;
ptrConfigPage^.wMaskBtPanelRight:=16#0;
ptrConfigPage^.wMaskFunctionPanel:=16#3F;
(* Navigation panel restriction *)
ptrConfigPage^.wMaskTouchScreenNavPanel:=16#3F;
(* Active machine movement mask *)
ptrConfigPage^.wMaskActiveMachineBtPanelLeft:=16#0;
ptrConfigPage^.wMaskActiveMachineBtPanelRight:=16#0;
ptrConfigPage^.wMaskActiveMachineFunctionPanel:=16#0;
ptrConfigPage^.wMaskActiveMachineNavPanel:=16#3F;
(* Button edge action *)
ptrConfigPage^.aiRTrigActionPanelRight[1]:=0;
ptrConfigPage^.aiRTrigActionPanelRight[2]:=0;
ptrConfigPage^.aiRTrigActionPanelRight[3]:=0;
ptrConfigPage^.aiRTrigActionPanelRight[4]:=0;
ptrConfigPage^.aiRTrigActionPanelRight[5]:=0;
ptrConfigPage^.aiFTrigActionPanelRight[1]:=0;
ptrConfigPage^.aiFTrigActionPanelRight[2]:=0;
ptrConfigPage^.aiFTrigActionPanelRight[3]:=0;
ptrConfigPage^.aiFTrigActionPanelRight[4]:=0;
ptrConfigPage^.aiFTrigActionPanelRight[5]:=0;
ptrConfigPage^.aiDelayActionPanelRight[1]:=0;
ptrConfigPage^.aiDelayActionPanelRight[2]:=0;
ptrConfigPage^.aiDelayActionPanelRight[3]:=0;
ptrConfigPage^.aiDelayActionPanelRight[4]:=0;
ptrConfigPage^.aiDelayActionPanelRight[5]:=0;
ptrConfigPage^.aiRTrigActionFunctionPanel[1]:=201;
ptrConfigPage^.aiRTrigActionFunctionPanel[2]:=202;
ptrConfigPage^.aiRTrigActionFunctionPanel[3]:=203;
ptrConfigPage^.aiRTrigActionFunctionPanel[4]:=204;
ptrConfigPage^.aiRTrigActionFunctionPanel[5]:=205;
ptrConfigPage^.aiRTrigActionFunctionPanel[6]:=1005;
ptrConfigPage^.aiRTrigActionFunctionPanel[7]:=0;
ptrConfigPage^.aiRTrigActionFunctionPanel[8]:=0;
ptrConfigPage^.aiRTrigActionFunctionPanel[9]:=0;
ptrConfigPage^.aiRTrigActionFunctionPanel[10]:=0;
ptrConfigPage^.aiRTrigActionFunctionPanel[11]:=0;
ptrConfigPage^.aiRTrigActionFunctionPanel[12]:=0;
ptrConfigPage^.aiFTrigActionTouchScreenNavPanel[1]:=10110;
ptrConfigPage^.aiFTrigActionTouchScreenNavPanel[2]:=10120;
ptrConfigPage^.aiFTrigActionTouchScreenNavPanel[3]:=10130;
ptrConfigPage^.aiFTrigActionTouchScreenNavPanel[4]:=10140;
ptrConfigPage^.aiFTrigActionTouchScreenNavPanel[5]:=10150;
ptrConfigPage^.aiFTrigActionTouchScreenNavPanel[6]:=10160;
ptrConfigPage^.xMaskBtStart:=FALSE;
ptrConfigPage^.xMaskBtStop:=TRUE;

(* QVis page 130, Profile *)
iIndexPage:=130;
iPageNumber:=iPageNumber+1;
T_Visu.T_PageIndex[iIndexPage].iIndexConfigPage:=iPageNumber;
ptrConfigPage:=ADR(T_Visu.T_ConfigPage[T_Visu.T_PageIndex[iIndexPage].iIndexConfigPage]);
ptrConfigPage^.sName:='Profile';
ptrConfigPage^.wMaskBtPanelLeft:=16#1F;
ptrConfigPage^.wMaskBtPanelRight:=16#E0;
ptrConfigPage^.wMaskFunctionPanel:=16#0;
(* Navigation panel restriction *)
ptrConfigPage^.wMaskTouchScreenNavPanel:=16#3F;
(* Active machine movement mask *)
ptrConfigPage^.wMaskActiveMachineBtPanelLeft:=16#0;
ptrConfigPage^.wMaskActiveMachineBtPanelRight:=16#0;
ptrConfigPage^.wMaskActiveMachineFunctionPanel:=16#0;
ptrConfigPage^.wMaskActiveMachineNavPanel:=16#3F;
(* Button edge action *)
ptrConfigPage^.aiRTrigActionPanelRight[1]:=1002;
ptrConfigPage^.aiRTrigActionPanelRight[2]:=1003;
ptrConfigPage^.aiRTrigActionPanelRight[3]:=1004;
ptrConfigPage^.aiRTrigActionPanelRight[4]:=0;
ptrConfigPage^.aiRTrigActionPanelRight[5]:=0;
ptrConfigPage^.aiFTrigActionPanelRight[1]:=0;
ptrConfigPage^.aiFTrigActionPanelRight[2]:=0;
ptrConfigPage^.aiFTrigActionPanelRight[3]:=0;
ptrConfigPage^.aiFTrigActionPanelRight[4]:=0;
ptrConfigPage^.aiFTrigActionPanelRight[5]:=0;
ptrConfigPage^.aiDelayActionPanelRight[1]:=0;
ptrConfigPage^.aiDelayActionPanelRight[2]:=0;
ptrConfigPage^.aiDelayActionPanelRight[3]:=0;
ptrConfigPage^.aiDelayActionPanelRight[4]:=0;
ptrConfigPage^.aiDelayActionPanelRight[5]:=0;
ptrConfigPage^.aiRTrigActionFunctionPanel[1]:=0;
ptrConfigPage^.aiRTrigActionFunctionPanel[2]:=0;
ptrConfigPage^.aiRTrigActionFunctionPanel[3]:=0;
ptrConfigPage^.aiRTrigActionFunctionPanel[4]:=0;
ptrConfigPage^.aiRTrigActionFunctionPanel[5]:=0;
ptrConfigPage^.aiRTrigActionFunctionPanel[6]:=0;
ptrConfigPage^.aiRTrigActionFunctionPanel[7]:=0;
ptrConfigPage^.aiRTrigActionFunctionPanel[8]:=0;
ptrConfigPage^.aiRTrigActionFunctionPanel[9]:=0;
ptrConfigPage^.aiRTrigActionFunctionPanel[10]:=0;
ptrConfigPage^.aiRTrigActionFunctionPanel[11]:=0;
ptrConfigPage^.aiRTrigActionFunctionPanel[12]:=0;
ptrConfigPage^.aiFTrigActionTouchScreenNavPanel[1]:=10110;
ptrConfigPage^.aiFTrigActionTouchScreenNavPanel[2]:=10120;
ptrConfigPage^.aiFTrigActionTouchScreenNavPanel[3]:=10130;
ptrConfigPage^.aiFTrigActionTouchScreenNavPanel[4]:=10140;
ptrConfigPage^.aiFTrigActionTouchScreenNavPanel[5]:=10150;
ptrConfigPage^.aiFTrigActionTouchScreenNavPanel[6]:=10160;
ptrConfigPage^.xMaskBtStart:=FALSE;
ptrConfigPage^.xMaskBtStop:=TRUE;

(* QVis page 140, General Setup *)
iIndexPage:=140;
iPageNumber:=iPageNumber+1;
T_Visu.T_PageIndex[iIndexPage].iIndexConfigPage:=iPageNumber;
ptrConfigPage:=ADR(T_Visu.T_ConfigPage[T_Visu.T_PageIndex[iIndexPage].iIndexConfigPage]);
ptrConfigPage^.sName:='General Setup';
ptrConfigPage^.wMaskBtPanelLeft:=16#1F;
ptrConfigPage^.wMaskBtPanelRight:=16#0;
ptrConfigPage^.wMaskFunctionPanel:=16#0;
(* Navigation panel restriction *)
ptrConfigPage^.wMaskTouchScreenNavPanel:=16#3F;
(* Active machine movement mask *)
ptrConfigPage^.wMaskActiveMachineBtPanelLeft:=16#0;
ptrConfigPage^.wMaskActiveMachineBtPanelRight:=16#0;
ptrConfigPage^.wMaskActiveMachineFunctionPanel:=16#0;
ptrConfigPage^.wMaskActiveMachineNavPanel:=16#3F;
(* Button edge action *)
ptrConfigPage^.aiRTrigActionPanelRight[1]:=0;
ptrConfigPage^.aiRTrigActionPanelRight[2]:=0;
ptrConfigPage^.aiRTrigActionPanelRight[3]:=0;
ptrConfigPage^.aiRTrigActionPanelRight[4]:=0;
ptrConfigPage^.aiRTrigActionPanelRight[5]:=0;
ptrConfigPage^.aiFTrigActionPanelRight[1]:=0;
ptrConfigPage^.aiFTrigActionPanelRight[2]:=0;
ptrConfigPage^.aiFTrigActionPanelRight[3]:=0;
ptrConfigPage^.aiFTrigActionPanelRight[4]:=0;
ptrConfigPage^.aiFTrigActionPanelRight[5]:=0;
ptrConfigPage^.aiDelayActionPanelRight[1]:=0;
ptrConfigPage^.aiDelayActionPanelRight[2]:=0;
ptrConfigPage^.aiDelayActionPanelRight[3]:=0;
ptrConfigPage^.aiDelayActionPanelRight[4]:=0;
ptrConfigPage^.aiDelayActionPanelRight[5]:=0;
ptrConfigPage^.aiRTrigActionFunctionPanel[1]:=0;
ptrConfigPage^.aiRTrigActionFunctionPanel[2]:=0;
ptrConfigPage^.aiRTrigActionFunctionPanel[3]:=0;
ptrConfigPage^.aiRTrigActionFunctionPanel[4]:=0;
ptrConfigPage^.aiRTrigActionFunctionPanel[5]:=0;
ptrConfigPage^.aiRTrigActionFunctionPanel[6]:=0;
ptrConfigPage^.aiRTrigActionFunctionPanel[7]:=0;
ptrConfigPage^.aiRTrigActionFunctionPanel[8]:=0;
ptrConfigPage^.aiRTrigActionFunctionPanel[9]:=0;
ptrConfigPage^.aiRTrigActionFunctionPanel[10]:=0;
ptrConfigPage^.aiRTrigActionFunctionPanel[11]:=0;
ptrConfigPage^.aiRTrigActionFunctionPanel[12]:=0;
ptrConfigPage^.aiFTrigActionTouchScreenNavPanel[1]:=10110;
ptrConfigPage^.aiFTrigActionTouchScreenNavPanel[2]:=10120;
ptrConfigPage^.aiFTrigActionTouchScreenNavPanel[3]:=10130;
ptrConfigPage^.aiFTrigActionTouchScreenNavPanel[4]:=10140;
ptrConfigPage^.aiFTrigActionTouchScreenNavPanel[5]:=10150;
ptrConfigPage^.aiFTrigActionTouchScreenNavPanel[6]:=10160;
ptrConfigPage^.xMaskBtStart:=FALSE;
ptrConfigPage^.xMaskBtStop:=TRUE;

(* QVis page 150, Configuration *)
iIndexPage:=150;
iPageNumber:=iPageNumber+1;
T_Visu.T_PageIndex[iIndexPage].iIndexConfigPage:=iPageNumber;
ptrConfigPage:=ADR(T_Visu.T_ConfigPage[T_Visu.T_PageIndex[iIndexPage].iIndexConfigPage]);
ptrConfigPage^.sName:='Configuration';
ptrConfigPage^.wMaskBtPanelLeft:=16#1F;
ptrConfigPage^.wMaskBtPanelRight:=16#0;
ptrConfigPage^.wMaskFunctionPanel:=16#0;
(* Navigation panel restriction *)
ptrConfigPage^.wMaskTouchScreenNavPanel:=16#3F;
(* Active machine movement mask *)
ptrConfigPage^.wMaskActiveMachineBtPanelLeft:=16#0;
ptrConfigPage^.wMaskActiveMachineBtPanelRight:=16#0;
ptrConfigPage^.wMaskActiveMachineFunctionPanel:=16#0;
ptrConfigPage^.wMaskActiveMachineNavPanel:=16#3F;
(* Button edge action *)
ptrConfigPage^.aiRTrigActionPanelRight[1]:=0;
ptrConfigPage^.aiRTrigActionPanelRight[2]:=0;
ptrConfigPage^.aiRTrigActionPanelRight[3]:=0;
ptrConfigPage^.aiRTrigActionPanelRight[4]:=0;
ptrConfigPage^.aiRTrigActionPanelRight[5]:=0;
ptrConfigPage^.aiFTrigActionPanelRight[1]:=0;
ptrConfigPage^.aiFTrigActionPanelRight[2]:=0;
ptrConfigPage^.aiFTrigActionPanelRight[3]:=0;
ptrConfigPage^.aiFTrigActionPanelRight[4]:=0;
ptrConfigPage^.aiFTrigActionPanelRight[5]:=0;
ptrConfigPage^.aiDelayActionPanelRight[1]:=0;
ptrConfigPage^.aiDelayActionPanelRight[2]:=0;
ptrConfigPage^.aiDelayActionPanelRight[3]:=0;
ptrConfigPage^.aiDelayActionPanelRight[4]:=0;
ptrConfigPage^.aiDelayActionPanelRight[5]:=0;
ptrConfigPage^.aiRTrigActionFunctionPanel[1]:=0;
ptrConfigPage^.aiRTrigActionFunctionPanel[2]:=0;
ptrConfigPage^.aiRTrigActionFunctionPanel[3]:=0;
ptrConfigPage^.aiRTrigActionFunctionPanel[4]:=0;
ptrConfigPage^.aiRTrigActionFunctionPanel[5]:=0;
ptrConfigPage^.aiRTrigActionFunctionPanel[6]:=0;
ptrConfigPage^.aiRTrigActionFunctionPanel[7]:=0;
ptrConfigPage^.aiRTrigActionFunctionPanel[8]:=0;
ptrConfigPage^.aiRTrigActionFunctionPanel[9]:=0;
ptrConfigPage^.aiRTrigActionFunctionPanel[10]:=0;
ptrConfigPage^.aiRTrigActionFunctionPanel[11]:=0;
ptrConfigPage^.aiRTrigActionFunctionPanel[12]:=0;
ptrConfigPage^.aiFTrigActionTouchScreenNavPanel[1]:=10110;
ptrConfigPage^.aiFTrigActionTouchScreenNavPanel[2]:=10120;
ptrConfigPage^.aiFTrigActionTouchScreenNavPanel[3]:=10130;
ptrConfigPage^.aiFTrigActionTouchScreenNavPanel[4]:=10140;
ptrConfigPage^.aiFTrigActionTouchScreenNavPanel[5]:=10150;
ptrConfigPage^.aiFTrigActionTouchScreenNavPanel[6]:=10160;
ptrConfigPage^.xMaskBtStart:=FALSE;
ptrConfigPage^.xMaskBtStop:=TRUE;

(* QVis page 160, Error List *)
iIndexPage:=160;
iPageNumber:=iPageNumber+1;
T_Visu.T_PageIndex[iIndexPage].iIndexConfigPage:=iPageNumber;
ptrConfigPage:=ADR(T_Visu.T_ConfigPage[T_Visu.T_PageIndex[iIndexPage].iIndexConfigPage]);
ptrConfigPage^.sName:='Error List';
ptrConfigPage^.wMaskBtPanelLeft:=16#1F;
ptrConfigPage^.wMaskBtPanelRight:=16#60;
ptrConfigPage^.wMaskFunctionPanel:=16#0;
(* Navigation panel restriction *)
ptrConfigPage^.wMaskTouchScreenNavPanel:=16#3F;
(* Active machine movement mask *)
ptrConfigPage^.wMaskActiveMachineBtPanelLeft:=16#0;
ptrConfigPage^.wMaskActiveMachineBtPanelRight:=16#60;
ptrConfigPage^.wMaskActiveMachineFunctionPanel:=16#0;
ptrConfigPage^.wMaskActiveMachineNavPanel:=16#3F;
(* Button edge action *)
ptrConfigPage^.aiRTrigActionPanelRight[1]:=99;
ptrConfigPage^.aiRTrigActionPanelRight[2]:=20;
ptrConfigPage^.aiRTrigActionPanelRight[3]:=0;
ptrConfigPage^.aiRTrigActionPanelRight[4]:=0;
ptrConfigPage^.aiRTrigActionPanelRight[5]:=0;
ptrConfigPage^.aiFTrigActionPanelRight[1]:=0;
ptrConfigPage^.aiFTrigActionPanelRight[2]:=0;
ptrConfigPage^.aiFTrigActionPanelRight[3]:=0;
ptrConfigPage^.aiFTrigActionPanelRight[4]:=0;
ptrConfigPage^.aiFTrigActionPanelRight[5]:=0;
ptrConfigPage^.aiDelayActionPanelRight[1]:=0;
ptrConfigPage^.aiDelayActionPanelRight[2]:=0;
ptrConfigPage^.aiDelayActionPanelRight[3]:=0;
ptrConfigPage^.aiDelayActionPanelRight[4]:=0;
ptrConfigPage^.aiDelayActionPanelRight[5]:=0;
ptrConfigPage^.aiRTrigActionFunctionPanel[1]:=0;
ptrConfigPage^.aiRTrigActionFunctionPanel[2]:=0;
ptrConfigPage^.aiRTrigActionFunctionPanel[3]:=0;
ptrConfigPage^.aiRTrigActionFunctionPanel[4]:=0;
ptrConfigPage^.aiRTrigActionFunctionPanel[5]:=0;
ptrConfigPage^.aiRTrigActionFunctionPanel[6]:=0;
ptrConfigPage^.aiRTrigActionFunctionPanel[7]:=0;
ptrConfigPage^.aiRTrigActionFunctionPanel[8]:=0;
ptrConfigPage^.aiRTrigActionFunctionPanel[9]:=0;
ptrConfigPage^.aiRTrigActionFunctionPanel[10]:=0;
ptrConfigPage^.aiRTrigActionFunctionPanel[11]:=0;
ptrConfigPage^.aiRTrigActionFunctionPanel[12]:=0;
ptrConfigPage^.aiFTrigActionTouchScreenNavPanel[1]:=10110;
ptrConfigPage^.aiFTrigActionTouchScreenNavPanel[2]:=10120;
ptrConfigPage^.aiFTrigActionTouchScreenNavPanel[3]:=10130;
ptrConfigPage^.aiFTrigActionTouchScreenNavPanel[4]:=10140;
ptrConfigPage^.aiFTrigActionTouchScreenNavPanel[5]:=10150;
ptrConfigPage^.aiFTrigActionTouchScreenNavPanel[6]:=10160;
ptrConfigPage^.xMaskBtStart:=FALSE;
ptrConfigPage^.xMaskBtStop:=TRUE;

(* QVis page 170, Parameter General *)
iIndexPage:=170;
iPageNumber:=iPageNumber+1;
T_Visu.T_PageIndex[iIndexPage].iIndexConfigPage:=iPageNumber;
ptrConfigPage:=ADR(T_Visu.T_ConfigPage[T_Visu.T_PageIndex[iIndexPage].iIndexConfigPage]);
ptrConfigPage^.sName:='Parameter General';
ptrConfigPage^.wMaskBtPanelLeft:=16#1F;
ptrConfigPage^.wMaskBtPanelRight:=16#200;
ptrConfigPage^.wMaskFunctionPanel:=16#0;
(* Navigation panel restriction *)
ptrConfigPage^.wMaskTouchScreenNavPanel:=16#3F;
(* Active machine movement mask *)
ptrConfigPage^.wMaskActiveMachineBtPanelLeft:=16#0;
ptrConfigPage^.wMaskActiveMachineBtPanelRight:=16#0;
ptrConfigPage^.wMaskActiveMachineFunctionPanel:=16#0;
ptrConfigPage^.wMaskActiveMachineNavPanel:=16#3F;
(* Button edge action *)
ptrConfigPage^.aiRTrigActionPanelRight[1]:=0;
ptrConfigPage^.aiRTrigActionPanelRight[2]:=0;
ptrConfigPage^.aiRTrigActionPanelRight[3]:=0;
ptrConfigPage^.aiRTrigActionPanelRight[4]:=0;
ptrConfigPage^.aiRTrigActionPanelRight[5]:=1006;
ptrConfigPage^.aiFTrigActionPanelRight[1]:=0;
ptrConfigPage^.aiFTrigActionPanelRight[2]:=0;
ptrConfigPage^.aiFTrigActionPanelRight[3]:=0;
ptrConfigPage^.aiFTrigActionPanelRight[4]:=0;
ptrConfigPage^.aiFTrigActionPanelRight[5]:=0;
ptrConfigPage^.aiDelayActionPanelRight[1]:=0;
ptrConfigPage^.aiDelayActionPanelRight[2]:=0;
ptrConfigPage^.aiDelayActionPanelRight[3]:=0;
ptrConfigPage^.aiDelayActionPanelRight[4]:=0;
ptrConfigPage^.aiDelayActionPanelRight[5]:=0;
ptrConfigPage^.aiRTrigActionFunctionPanel[1]:=0;
ptrConfigPage^.aiRTrigActionFunctionPanel[2]:=0;
ptrConfigPage^.aiRTrigActionFunctionPanel[3]:=0;
ptrConfigPage^.aiRTrigActionFunctionPanel[4]:=0;
ptrConfigPage^.aiRTrigActionFunctionPanel[5]:=0;
ptrConfigPage^.aiRTrigActionFunctionPanel[6]:=0;
ptrConfigPage^.aiRTrigActionFunctionPanel[7]:=0;
ptrConfigPage^.aiRTrigActionFunctionPanel[8]:=0;
ptrConfigPage^.aiRTrigActionFunctionPanel[9]:=0;
ptrConfigPage^.aiRTrigActionFunctionPanel[10]:=0;
ptrConfigPage^.aiRTrigActionFunctionPanel[11]:=0;
ptrConfigPage^.aiRTrigActionFunctionPanel[12]:=0;
ptrConfigPage^.aiFTrigActionTouchScreenNavPanel[1]:=10110;
ptrConfigPage^.aiFTrigActionTouchScreenNavPanel[2]:=10120;
ptrConfigPage^.aiFTrigActionTouchScreenNavPanel[3]:=10130;
ptrConfigPage^.aiFTrigActionTouchScreenNavPanel[4]:=10140;
ptrConfigPage^.aiFTrigActionTouchScreenNavPanel[5]:=10150;
ptrConfigPage^.aiFTrigActionTouchScreenNavPanel[6]:=10160;
ptrConfigPage^.xMaskBtStart:=FALSE;
ptrConfigPage^.xMaskBtStop:=TRUE;

(* QVis page 210, Teach-in Tool Rotation *)
iIndexPage:=210;
iPageNumber:=iPageNumber+1;
T_Visu.T_PageIndex[iIndexPage].iIndexConfigPage:=iPageNumber;
ptrConfigPage:=ADR(T_Visu.T_ConfigPage[T_Visu.T_PageIndex[iIndexPage].iIndexConfigPage]);
ptrConfigPage^.sName:='Teach-in Tool Rotation';
ptrConfigPage^.wMaskBtPanelLeft:=16#1F;
ptrConfigPage^.wMaskBtPanelRight:=16#1E0;
ptrConfigPage^.wMaskFunctionPanel:=16#F;
(* Navigation panel restriction *)
ptrConfigPage^.wMaskTouchScreenNavPanel:=16#27;
(* Active machine movement mask *)
ptrConfigPage^.wMaskActiveMachineBtPanelLeft:=16#0;
ptrConfigPage^.wMaskActiveMachineBtPanelRight:=16#0;
ptrConfigPage^.wMaskActiveMachineFunctionPanel:=16#0;
ptrConfigPage^.wMaskActiveMachineNavPanel:=16#27;
(* Button edge action *)
ptrConfigPage^.aiRTrigActionPanelRight[1]:=312;
ptrConfigPage^.aiRTrigActionPanelRight[2]:=310;
ptrConfigPage^.aiRTrigActionPanelRight[3]:=316;
ptrConfigPage^.aiRTrigActionPanelRight[4]:=314;
ptrConfigPage^.aiRTrigActionPanelRight[5]:=0;
ptrConfigPage^.aiFTrigActionPanelRight[1]:=0;
ptrConfigPage^.aiFTrigActionPanelRight[2]:=0;
ptrConfigPage^.aiFTrigActionPanelRight[3]:=301;
ptrConfigPage^.aiFTrigActionPanelRight[4]:=301;
ptrConfigPage^.aiFTrigActionPanelRight[5]:=0;
ptrConfigPage^.aiDelayActionPanelRight[1]:=0;
ptrConfigPage^.aiDelayActionPanelRight[2]:=0;
ptrConfigPage^.aiDelayActionPanelRight[3]:=0;
ptrConfigPage^.aiDelayActionPanelRight[4]:=0;
ptrConfigPage^.aiDelayActionPanelRight[5]:=0;
ptrConfigPage^.aiRTrigActionFunctionPanel[1]:=322;
ptrConfigPage^.aiRTrigActionFunctionPanel[2]:=323;
ptrConfigPage^.aiRTrigActionFunctionPanel[3]:=321;
ptrConfigPage^.aiRTrigActionFunctionPanel[4]:=320;
ptrConfigPage^.aiRTrigActionFunctionPanel[5]:=0;
ptrConfigPage^.aiRTrigActionFunctionPanel[6]:=0;
ptrConfigPage^.aiRTrigActionFunctionPanel[7]:=0;
ptrConfigPage^.aiRTrigActionFunctionPanel[8]:=0;
ptrConfigPage^.aiRTrigActionFunctionPanel[9]:=0;
ptrConfigPage^.aiRTrigActionFunctionPanel[10]:=0;
ptrConfigPage^.aiRTrigActionFunctionPanel[11]:=0;
ptrConfigPage^.aiRTrigActionFunctionPanel[12]:=0;
ptrConfigPage^.aiFTrigActionTouchScreenNavPanel[1]:=10210;
ptrConfigPage^.aiFTrigActionTouchScreenNavPanel[2]:=10220;
ptrConfigPage^.aiFTrigActionTouchScreenNavPanel[3]:=10230;
ptrConfigPage^.aiFTrigActionTouchScreenNavPanel[4]:=0;
ptrConfigPage^.aiFTrigActionTouchScreenNavPanel[5]:=0;
ptrConfigPage^.aiFTrigActionTouchScreenNavPanel[6]:=10260;
ptrConfigPage^.xMaskBtStart:=TRUE;
ptrConfigPage^.xMaskBtStop:=TRUE;

(* QVis page 220, Tool Torque *)
iIndexPage:=220;
iPageNumber:=iPageNumber+1;
T_Visu.T_PageIndex[iIndexPage].iIndexConfigPage:=iPageNumber;
ptrConfigPage:=ADR(T_Visu.T_ConfigPage[T_Visu.T_PageIndex[iIndexPage].iIndexConfigPage]);
ptrConfigPage^.sName:='Tool Torque';
ptrConfigPage^.wMaskBtPanelLeft:=16#1F;
ptrConfigPage^.wMaskBtPanelRight:=16#0;
ptrConfigPage^.wMaskFunctionPanel:=16#DF;
(* Navigation panel restriction *)
ptrConfigPage^.wMaskTouchScreenNavPanel:=16#27;
(* Active machine movement mask *)
ptrConfigPage^.wMaskActiveMachineBtPanelLeft:=16#0;
ptrConfigPage^.wMaskActiveMachineBtPanelRight:=16#0;
ptrConfigPage^.wMaskActiveMachineFunctionPanel:=16#DF;
ptrConfigPage^.wMaskActiveMachineNavPanel:=16#27;
(* Button edge action *)
ptrConfigPage^.aiRTrigActionPanelRight[1]:=0;
ptrConfigPage^.aiRTrigActionPanelRight[2]:=0;
ptrConfigPage^.aiRTrigActionPanelRight[3]:=0;
ptrConfigPage^.aiRTrigActionPanelRight[4]:=0;
ptrConfigPage^.aiRTrigActionPanelRight[5]:=0;
ptrConfigPage^.aiFTrigActionPanelRight[1]:=0;
ptrConfigPage^.aiFTrigActionPanelRight[2]:=0;
ptrConfigPage^.aiFTrigActionPanelRight[3]:=0;
ptrConfigPage^.aiFTrigActionPanelRight[4]:=0;
ptrConfigPage^.aiFTrigActionPanelRight[5]:=0;
ptrConfigPage^.aiDelayActionPanelRight[1]:=0;
ptrConfigPage^.aiDelayActionPanelRight[2]:=0;
ptrConfigPage^.aiDelayActionPanelRight[3]:=0;
ptrConfigPage^.aiDelayActionPanelRight[4]:=0;
ptrConfigPage^.aiDelayActionPanelRight[5]:=0;
ptrConfigPage^.aiRTrigActionFunctionPanel[1]:=502;
ptrConfigPage^.aiRTrigActionFunctionPanel[2]:=503;
ptrConfigPage^.aiRTrigActionFunctionPanel[3]:=501;
ptrConfigPage^.aiRTrigActionFunctionPanel[4]:=130;
ptrConfigPage^.aiRTrigActionFunctionPanel[5]:=131;
ptrConfigPage^.aiRTrigActionFunctionPanel[6]:=0;
ptrConfigPage^.aiRTrigActionFunctionPanel[7]:=504;
ptrConfigPage^.aiRTrigActionFunctionPanel[8]:=505;
ptrConfigPage^.aiRTrigActionFunctionPanel[9]:=0;
ptrConfigPage^.aiRTrigActionFunctionPanel[10]:=0;
ptrConfigPage^.aiRTrigActionFunctionPanel[11]:=0;
ptrConfigPage^.aiRTrigActionFunctionPanel[12]:=0;
ptrConfigPage^.aiFTrigActionTouchScreenNavPanel[1]:=10210;
ptrConfigPage^.aiFTrigActionTouchScreenNavPanel[2]:=10220;
ptrConfigPage^.aiFTrigActionTouchScreenNavPanel[3]:=10230;
ptrConfigPage^.aiFTrigActionTouchScreenNavPanel[4]:=0;
ptrConfigPage^.aiFTrigActionTouchScreenNavPanel[5]:=0;
ptrConfigPage^.aiFTrigActionTouchScreenNavPanel[6]:=10260;
ptrConfigPage^.xMaskBtStart:=TRUE;
ptrConfigPage^.xMaskBtStop:=TRUE;

(* QVis page 230, Tool Tension *)
iIndexPage:=230;
iPageNumber:=iPageNumber+1;
T_Visu.T_PageIndex[iIndexPage].iIndexConfigPage:=iPageNumber;
ptrConfigPage:=ADR(T_Visu.T_ConfigPage[T_Visu.T_PageIndex[iIndexPage].iIndexConfigPage]);
ptrConfigPage^.sName:='Tool Tension';
ptrConfigPage^.wMaskBtPanelLeft:=16#1F;
ptrConfigPage^.wMaskBtPanelRight:=16#20;
ptrConfigPage^.wMaskFunctionPanel:=16#0;
(* Navigation panel restriction *)
ptrConfigPage^.wMaskTouchScreenNavPanel:=16#27;
(* Active machine movement mask *)
ptrConfigPage^.wMaskActiveMachineBtPanelLeft:=16#0;
ptrConfigPage^.wMaskActiveMachineBtPanelRight:=16#0;
ptrConfigPage^.wMaskActiveMachineFunctionPanel:=16#0;
ptrConfigPage^.wMaskActiveMachineNavPanel:=16#27;
(* Button edge action *)
ptrConfigPage^.aiRTrigActionPanelRight[1]:=501;
ptrConfigPage^.aiRTrigActionPanelRight[2]:=0;
ptrConfigPage^.aiRTrigActionPanelRight[3]:=0;
ptrConfigPage^.aiRTrigActionPanelRight[4]:=0;
ptrConfigPage^.aiRTrigActionPanelRight[5]:=0;
ptrConfigPage^.aiFTrigActionPanelRight[1]:=0;
ptrConfigPage^.aiFTrigActionPanelRight[2]:=0;
ptrConfigPage^.aiFTrigActionPanelRight[3]:=0;
ptrConfigPage^.aiFTrigActionPanelRight[4]:=0;
ptrConfigPage^.aiFTrigActionPanelRight[5]:=0;
ptrConfigPage^.aiDelayActionPanelRight[1]:=0;
ptrConfigPage^.aiDelayActionPanelRight[2]:=0;
ptrConfigPage^.aiDelayActionPanelRight[3]:=0;
ptrConfigPage^.aiDelayActionPanelRight[4]:=0;
ptrConfigPage^.aiDelayActionPanelRight[5]:=0;
ptrConfigPage^.aiRTrigActionFunctionPanel[1]:=0;
ptrConfigPage^.aiRTrigActionFunctionPanel[2]:=0;
ptrConfigPage^.aiRTrigActionFunctionPanel[3]:=0;
ptrConfigPage^.aiRTrigActionFunctionPanel[4]:=0;
ptrConfigPage^.aiRTrigActionFunctionPanel[5]:=0;
ptrConfigPage^.aiRTrigActionFunctionPanel[6]:=0;
ptrConfigPage^.aiRTrigActionFunctionPanel[7]:=0;
ptrConfigPage^.aiRTrigActionFunctionPanel[8]:=0;
ptrConfigPage^.aiRTrigActionFunctionPanel[9]:=0;
ptrConfigPage^.aiRTrigActionFunctionPanel[10]:=0;
ptrConfigPage^.aiRTrigActionFunctionPanel[11]:=0;
ptrConfigPage^.aiRTrigActionFunctionPanel[12]:=0;
ptrConfigPage^.aiFTrigActionTouchScreenNavPanel[1]:=10210;
ptrConfigPage^.aiFTrigActionTouchScreenNavPanel[2]:=10220;
ptrConfigPage^.aiFTrigActionTouchScreenNavPanel[3]:=10230;
ptrConfigPage^.aiFTrigActionTouchScreenNavPanel[4]:=0;
ptrConfigPage^.aiFTrigActionTouchScreenNavPanel[5]:=0;
ptrConfigPage^.aiFTrigActionTouchScreenNavPanel[6]:=10260;
ptrConfigPage^.xMaskBtStart:=FALSE;
ptrConfigPage^.xMaskBtStop:=TRUE;

(* QVis page 260, Error List *)
iIndexPage:=260;
iPageNumber:=iPageNumber+1;
T_Visu.T_PageIndex[iIndexPage].iIndexConfigPage:=iPageNumber;
ptrConfigPage:=ADR(T_Visu.T_ConfigPage[T_Visu.T_PageIndex[iIndexPage].iIndexConfigPage]);
ptrConfigPage^.sName:='Error List';
ptrConfigPage^.wMaskBtPanelLeft:=16#1F;
ptrConfigPage^.wMaskBtPanelRight:=16#60;
ptrConfigPage^.wMaskFunctionPanel:=16#0;
(* Navigation panel restriction *)
ptrConfigPage^.wMaskTouchScreenNavPanel:=16#27;
(* Active machine movement mask *)
ptrConfigPage^.wMaskActiveMachineBtPanelLeft:=16#0;
ptrConfigPage^.wMaskActiveMachineBtPanelRight:=16#60;
ptrConfigPage^.wMaskActiveMachineFunctionPanel:=16#0;
ptrConfigPage^.wMaskActiveMachineNavPanel:=16#27;
(* Button edge action *)
ptrConfigPage^.aiRTrigActionPanelRight[1]:=99;
ptrConfigPage^.aiRTrigActionPanelRight[2]:=20;
ptrConfigPage^.aiRTrigActionPanelRight[3]:=0;
ptrConfigPage^.aiRTrigActionPanelRight[4]:=0;
ptrConfigPage^.aiRTrigActionPanelRight[5]:=0;
ptrConfigPage^.aiFTrigActionPanelRight[1]:=0;
ptrConfigPage^.aiFTrigActionPanelRight[2]:=0;
ptrConfigPage^.aiFTrigActionPanelRight[3]:=0;
ptrConfigPage^.aiFTrigActionPanelRight[4]:=0;
ptrConfigPage^.aiFTrigActionPanelRight[5]:=0;
ptrConfigPage^.aiDelayActionPanelRight[1]:=0;
ptrConfigPage^.aiDelayActionPanelRight[2]:=0;
ptrConfigPage^.aiDelayActionPanelRight[3]:=0;
ptrConfigPage^.aiDelayActionPanelRight[4]:=0;
ptrConfigPage^.aiDelayActionPanelRight[5]:=0;
ptrConfigPage^.aiRTrigActionFunctionPanel[1]:=0;
ptrConfigPage^.aiRTrigActionFunctionPanel[2]:=0;
ptrConfigPage^.aiRTrigActionFunctionPanel[3]:=0;
ptrConfigPage^.aiRTrigActionFunctionPanel[4]:=0;
ptrConfigPage^.aiRTrigActionFunctionPanel[5]:=0;
ptrConfigPage^.aiRTrigActionFunctionPanel[6]:=0;
ptrConfigPage^.aiRTrigActionFunctionPanel[7]:=0;
ptrConfigPage^.aiRTrigActionFunctionPanel[8]:=0;
ptrConfigPage^.aiRTrigActionFunctionPanel[9]:=0;
ptrConfigPage^.aiRTrigActionFunctionPanel[10]:=0;
ptrConfigPage^.aiRTrigActionFunctionPanel[11]:=0;
ptrConfigPage^.aiRTrigActionFunctionPanel[12]:=0;
ptrConfigPage^.aiFTrigActionTouchScreenNavPanel[1]:=10210;
ptrConfigPage^.aiFTrigActionTouchScreenNavPanel[2]:=10220;
ptrConfigPage^.aiFTrigActionTouchScreenNavPanel[3]:=10230;
ptrConfigPage^.aiFTrigActionTouchScreenNavPanel[4]:=0;
ptrConfigPage^.aiFTrigActionTouchScreenNavPanel[5]:=0;
ptrConfigPage^.aiFTrigActionTouchScreenNavPanel[6]:=10260;
ptrConfigPage^.xMaskBtStart:=FALSE;
ptrConfigPage^.xMaskBtStop:=TRUE;

(* QVis page 270, Parameter Tool Rotation *)
iIndexPage:=270;
iPageNumber:=iPageNumber+1;
T_Visu.T_PageIndex[iIndexPage].iIndexConfigPage:=iPageNumber;
ptrConfigPage:=ADR(T_Visu.T_ConfigPage[T_Visu.T_PageIndex[iIndexPage].iIndexConfigPage]);
ptrConfigPage^.sName:='Parameter Tool Rotation';
ptrConfigPage^.wMaskBtPanelLeft:=16#1F;
ptrConfigPage^.wMaskBtPanelRight:=16#200;
ptrConfigPage^.wMaskFunctionPanel:=16#0;
(* Navigation panel restriction *)
ptrConfigPage^.wMaskTouchScreenNavPanel:=16#27;
(* Active machine movement mask *)
ptrConfigPage^.wMaskActiveMachineBtPanelLeft:=16#0;
ptrConfigPage^.wMaskActiveMachineBtPanelRight:=16#0;
ptrConfigPage^.wMaskActiveMachineFunctionPanel:=16#0;
ptrConfigPage^.wMaskActiveMachineNavPanel:=16#27;
(* Button edge action *)
ptrConfigPage^.aiRTrigActionPanelRight[1]:=0;
ptrConfigPage^.aiRTrigActionPanelRight[2]:=0;
ptrConfigPage^.aiRTrigActionPanelRight[3]:=0;
ptrConfigPage^.aiRTrigActionPanelRight[4]:=0;
ptrConfigPage^.aiRTrigActionPanelRight[5]:=1006;
ptrConfigPage^.aiFTrigActionPanelRight[1]:=0;
ptrConfigPage^.aiFTrigActionPanelRight[2]:=0;
ptrConfigPage^.aiFTrigActionPanelRight[3]:=0;
ptrConfigPage^.aiFTrigActionPanelRight[4]:=0;
ptrConfigPage^.aiFTrigActionPanelRight[5]:=0;
ptrConfigPage^.aiDelayActionPanelRight[1]:=0;
ptrConfigPage^.aiDelayActionPanelRight[2]:=0;
ptrConfigPage^.aiDelayActionPanelRight[3]:=0;
ptrConfigPage^.aiDelayActionPanelRight[4]:=0;
ptrConfigPage^.aiDelayActionPanelRight[5]:=0;
ptrConfigPage^.aiRTrigActionFunctionPanel[1]:=0;
ptrConfigPage^.aiRTrigActionFunctionPanel[2]:=0;
ptrConfigPage^.aiRTrigActionFunctionPanel[3]:=0;
ptrConfigPage^.aiRTrigActionFunctionPanel[4]:=0;
ptrConfigPage^.aiRTrigActionFunctionPanel[5]:=0;
ptrConfigPage^.aiRTrigActionFunctionPanel[6]:=0;
ptrConfigPage^.aiRTrigActionFunctionPanel[7]:=0;
ptrConfigPage^.aiRTrigActionFunctionPanel[8]:=0;
ptrConfigPage^.aiRTrigActionFunctionPanel[9]:=0;
ptrConfigPage^.aiRTrigActionFunctionPanel[10]:=0;
ptrConfigPage^.aiRTrigActionFunctionPanel[11]:=0;
ptrConfigPage^.aiRTrigActionFunctionPanel[12]:=0;
ptrConfigPage^.aiFTrigActionTouchScreenNavPanel[1]:=10210;
ptrConfigPage^.aiFTrigActionTouchScreenNavPanel[2]:=10220;
ptrConfigPage^.aiFTrigActionTouchScreenNavPanel[3]:=10230;
ptrConfigPage^.aiFTrigActionTouchScreenNavPanel[4]:=0;
ptrConfigPage^.aiFTrigActionTouchScreenNavPanel[5]:=0;
ptrConfigPage^.aiFTrigActionTouchScreenNavPanel[6]:=10260;
ptrConfigPage^.xMaskBtStart:=FALSE;
ptrConfigPage^.xMaskBtStop:=TRUE;

